C07247=1066.189,109.363,-74.257,172.619,27.910,155.103
C07248=1066.184,109.114,-74.238,172.618,27.907,155.103
C07249=1066.178,108.864,-74.219,172.616,27.904,155.103
C07250=1066.172,108.615,-74.200,172.615,27.901,155.102
C07251=1066.166,108.366,-74.181,172.613,27.898,155.102
C07252=1066.160,108.117,-74.161,172.612,27.896,155.101
C07253=1066.154,107.868,-74.142,172.609,27.893,155.101
C07254=1066.148,107.618,-74.123,172.608,27.890,155.101
C07255=1066.143,107.370,-74.104,172.606,27.887,155.100
C07256=1066.137,107.120,-74.085,172.604,27.885,155.100
C07257=1066.131,106.871,-74.066,172.603,27.882,155.100
C07258=1066.125,106.621,-74.047,172.601,27.879,155.099
C07259=1066.119,106.373,-74.027,172.600,27.877,155.099
C07260=1066.113,106.123,-74.008,172.598,27.874,155.098
C07261=1066.107,105.874,-73.989,172.597,27.871,155.098
C07262=1066.102,105.625,-73.969,172.595,27.868,155.098
C07263=1066.096,105.376,-73.951,172.594,27.865,155.097
C07264=1066.090,105.127,-73.932,172.592,27.863,155.097
C07265=1066.084,104.877,-73.913,172.591,27.860,155.096
C07266=1066.078,104.628,-73.894,172.589,27.857,155.096
C07267=1066.072,104.379,-73.875,172.588,27.854,155.095
C07268=1066.067,104.129,-73.856,172.586,27.852,155.095
C07269=1066.061,103.880,-73.836,172.584,27.849,155.095
C07270=1066.055,103.631,-73.818,172.583,27.847,155.094
C07271=1066.049,103.382,-73.799,172.581,27.844,155.094
C07272=1066.044,103.133,-73.779,172.580,27.841,155.094
C07273=1066.037,102.883,-73.761,172.579,27.838,155.093
C07274=1066.032,102.634,-73.742,172.578,27.836,155.093
C07275=1066.027,102.385,-73.723,172.576,27.833,155.092
C07276=1066.021,102.136,-73.703,172.575,27.830,155.092
C07277=1066.014,101.887,-73.685,172.573,27.827,155.092
C07278=1066.009,101.637,-73.666,172.572,27.825,155.091
C07279=1066.003,101.388,-73.646,172.570,27.822,155.091
C07280=1065.997,101.139,-73.628,172.568,27.819,155.090
C07281=1065.992,100.890,-73.609,172.567,27.816,155.090
C07282=1065.985,100.641,-73.590,172.565,27.813,155.090
C07283=1065.979,100.391,-73.571,172.564,27.811,155.089
C07284=1065.973,100.142,-73.552,172.562,27.808,155.089
C07285=1065.967,99.893,-73.533,172.561,27.806,155.088
C07286=1065.962,99.645,-73.515,172.559,27.803,155.088
C07287=1065.956,99.394,-73.496,172.558,27.800,155.088
C07288=1065.950,99.145,-73.478,172.556,27.797,155.087
C07289=1065.944,98.896,-73.458,172.555,27.794,155.087
C07290=1065.938,98.647,-73.440,172.553,27.792,155.086
C07291=1065.933,98.398,-73.421,172.551,27.789,155.086
C07292=1065.926,98.149,-73.402,172.550,27.787,155.086
C07293=1065.921,97.899,-73.384,172.548,27.784,155.085
C07294=1065.914,97.650,-73.365,172.547,27.781,155.085
C07295=1065.909,97.400,-73.346,172.545,27.778,155.085
C07296=1065.903,97.152,-73.327,172.544,27.775,155.084
C07297=1065.897,96.902,-73.308,172.542,27.773,155.084
C07298=1065.891,96.653,-73.290,172.541,27.770,155.083
C07299=1065.885,96.404,-73.272,172.539,27.767,155.083
C07300=1065.879,96.155,-73.253,172.538,27.765,155.083
C07301=1065.873,95.906,-73.234,172.536,27.762,155.082
C07302=1065.868,95.656,-73.216,172.535,27.759,155.082
C07303=1065.861,95.407,-73.197,172.533,27.756,155.081
C07304=1065.856,95.158,-73.178,172.531,27.754,155.081
C07305=1065.849,94.874,-73.157,172.530,27.751,155.081
C07306=1065.843,94.591,-73.136,172.529,27.748,155.080
C07307=1065.836,94.307,-73.115,172.526,27.745,155.080
C07308=1065.829,94.023,-73.094,172.525,27.741,155.079
C07309=1065.823,93.775,-73.075,172.523,27.738,155.079
C07310=1065.817,93.525,-73.057,172.522,27.736,155.078
C07311=1065.812,93.275,-73.038,172.520,27.733,155.078
C07312=1065.806,93.027,-73.019,172.519,27.730,155.078
C07313=1065.800,92.777,-73.001,172.517,27.728,155.077
C07314=1065.794,92.528,-72.982,172.515,27.725,155.077
C07315=1065.788,92.279,-72.964,172.514,27.722,155.077
C07316=1065.783,92.029,-72.945,172.512,27.719,155.076
C07317=1065.776,91.780,-72.927,172.511,27.717,155.076
C07318=1065.772,91.531,-72.909,172.510,27.714,155.075
C07319=1065.765,91.282,-72.890,172.509,27.711,155.075
C07320=1065.759,91.033,-72.871,172.507,27.708,155.075
C07321=1065.754,90.783,-72.853,172.506,27.706,155.074
C07322=1065.748,90.534,-72.834,172.504,27.703,155.074
C07323=1065.741,90.284,-72.816,172.503,27.700,155.073
C07324=1065.736,90.036,-72.798,172.501,27.697,155.073
C07325=1065.730,89.786,-72.780,172.499,27.695,155.073
C07326=1065.724,89.537,-72.761,172.498,27.692,155.072
C07327=1065.717,89.288,-72.742,172.496,27.689,155.072
C07328=1065.712,89.039,-72.725,172.495,27.687,155.071
C07329=1065.705,88.790,-72.706,172.493,27.684,155.071
C07330=1065.700,88.540,-72.688,172.492,27.681,155.071
C07331=1065.694,88.291,-72.669,172.490,27.679,155.070
C07332=1065.688,88.041,-72.651,172.489,27.676,155.070
C07333=1065.682,87.792,-72.633,172.487,27.673,155.070
C07334=1065.676,87.543,-72.615,172.486,27.670,155.069
C07335=1065.670,87.293,-72.597,172.484,27.668,155.069
C07336=1065.664,87.044,-72.578,172.483,27.665,155.068
C07337=1065.659,86.795,-72.560,172.481,27.663,155.068
C07338=1065.652,86.546,-72.542,172.480,27.660,155.068
C07339=1065.647,86.297,-72.524,172.478,27.657,155.067
C07340=1065.640,86.048,-72.506,172.476,27.654,155.067
C07341=1065.634,85.798,-72.488,172.476,27.652,155.066
C07342=1065.629,85.549,-72.470,172.474,27.649,155.066
C07343=1065.623,85.299,-72.451,172.473,27.646,155.066
C07344=1065.617,85.050,-72.433,172.471,27.643,155.065
C07345=1065.611,84.801,-72.415,172.470,27.641,155.065
C07346=1065.605,84.552,-72.397,172.468,27.638,155.065
C07347=1065.600,84.303,-72.379,172.467,27.635,155.064
C07348=1065.593,84.053,-72.360,172.465,27.633,155.064
C07349=1065.588,83.804,-72.343,172.464,27.630,155.063
C07350=1065.582,83.554,-72.324,172.462,27.627,155.063
C07351=1065.576,83.305,-72.306,172.461,27.624,155.063
C07352=1065.570,83.056,-72.288,172.459,27.621,155.062
C07353=1065.564,82.806,-72.270,172.458,27.619,155.062
C07354=1065.558,82.558,-72.252,172.456,27.616,155.062
C07355=1065.552,82.308,-72.234,172.454,27.614,155.061
C07356=1065.547,82.059,-72.216,172.453,27.611,155.061
C07357=1065.541,81.809,-72.199,172.451,27.608,155.060
C07358=1065.535,81.561,-72.180,172.451,27.605,155.060
C07359=1065.529,81.311,-72.162,172.449,27.603,155.059
C07360=1065.523,81.061,-72.144,172.448,27.600,155.059
C07361=1065.517,80.813,-72.125,172.446,27.597,155.059
C07362=1065.511,80.563,-72.108,172.445,27.594,155.058
C07363=1065.506,80.314,-72.090,172.443,27.591,155.058
C07364=1065.500,80.064,-72.072,172.442,27.589,155.058
C07365=1065.494,79.815,-72.054,172.440,27.586,155.057
C07366=1065.488,79.566,-72.036,172.439,27.583,155.057
C07367=1065.482,79.317,-72.018,172.437,27.581,155.056
C07368=1065.476,79.067,-72.000,172.436,27.578,155.056
C07369=1065.470,78.784,-71.980,172.434,27.575,155.056
C07370=1065.464,78.500,-71.960,172.433,27.572,155.055
C07371=1065.456,78.217,-71.940,172.431,27.568,155.055
C07372=1065.449,77.933,-71.919,172.429,27.565,155.054
C07373=1065.444,77.684,-71.901,172.427,27.563,155.054
C07374=1065.438,77.435,-71.883,172.427,27.560,155.053
C07375=1065.432,77.186,-71.866,172.425,27.557,155.053
C07376=1065.426,76.936,-71.848,172.424,27.555,155.053
C07377=1065.420,76.687,-71.831,172.422,27.552,155.052
C07378=1065.414,76.437,-71.813,172.421,27.549,155.052
C07379=1065.408,76.189,-71.795,172.419,27.547,155.052
C07380=1065.402,75.939,-71.777,172.418,27.544,155.051
C07381=1065.396,75.690,-71.759,172.416,27.541,155.051
C07382=1065.390,75.440,-71.741,172.415,27.539,155.050
C07383=1065.385,75.191,-71.724,172.413,27.536,155.050
C07384=1065.379,74.942,-71.706,172.412,27.533,155.050
C07385=1065.372,74.693,-71.689,172.410,27.530,155.049
C07386=1065.366,74.443,-71.671,172.409,27.527,155.049
C07387=1065.361,74.194,-71.653,172.407,27.525,155.048
C07388=1065.355,73.944,-71.635,172.406,27.522,155.048
C07389=1065.349,73.695,-71.618,172.405,27.520,155.048
C07390=1065.343,73.446,-71.600,172.403,27.517,155.047
C07391=1065.337,73.197,-71.583,172.402,27.514,155.047
C07392=1065.331,72.948,-71.565,172.400,27.511,155.047
C07393=1065.325,72.698,-71.547,172.399,27.509,155.046
C07394=1065.320,72.449,-71.530,172.397,27.506,155.046
C07395=1065.313,72.199,-71.512,172.396,27.503,155.045
C07396=1065.308,71.950,-71.494,172.394,27.500,155.045
C07397=1065.301,71.701,-71.477,172.393,27.498,155.045
C07398=1065.296,71.452,-71.459,172.391,27.495,155.044
C07399=1065.290,71.203,-71.442,172.390,27.492,155.044
C07400=1065.284,70.953,-71.424,172.388,27.489,155.043
C07401=1065.279,70.703,-71.407,172.388,27.487,155.043
C07402=1065.272,70.454,-71.390,172.386,27.484,155.043
C07403=1065.266,70.205,-71.372,172.385,27.481,155.042
C07404=1065.261,69.956,-71.354,172.383,27.479,155.042
C07405=1065.255,69.706,-71.336,172.382,27.476,155.042
C07406=1065.248,69.457,-71.319,172.380,27.473,155.041
C07407=1065.242,69.208,-71.302,172.379,27.471,155.041
C07408=1065.237,68.959,-71.284,172.377,27.468,155.040
C07409=1065.230,68.708,-71.267,172.376,27.465,155.040
C07410=1065.225,68.459,-71.250,172.374,27.463,155.040
C07411=1065.219,68.210,-71.232,172.372,27.460,155.039
C07412=1065.212,67.961,-71.215,172.371,27.457,155.039
C07413=1065.207,67.712,-71.197,172.369,27.454,155.039
C07414=1065.202,67.462,-71.180,172.369,27.452,155.038
C07415=1065.195,67.213,-71.163,172.367,27.449,155.038
C07416=1065.189,66.964,-71.146,172.366,27.447,155.037
C07417=1065.183,66.714,-71.128,172.364,27.444,155.037
C07418=1065.177,66.465,-71.111,172.363,27.441,155.037
C07419=1065.172,66.216,-71.094,172.361,27.438,155.036
C07420=1065.165,65.966,-71.076,172.360,27.435,155.036
C07421=1065.159,65.717,-71.059,172.358,27.433,155.035
C07422=1065.154,65.468,-71.041,172.357,27.430,155.035
C07423=1065.147,65.218,-71.025,172.355,27.428,155.035
C07424=1065.142,64.969,-71.007,172.354,27.425,155.034
C07425=1065.136,64.720,-70.990,172.352,27.422,155.034
C07426=1065.130,64.470,-70.973,172.352,27.419,155.034
C07427=1065.124,64.221,-70.955,172.350,27.417,155.033
C07428=1065.117,63.972,-70.938,172.349,27.414,155.033
C07429=1065.111,63.722,-70.922,172.347,27.411,155.032
C07430=1065.106,63.473,-70.904,172.346,27.409,155.032
C07431=1065.099,63.224,-70.887,172.344,27.406,155.032
C07432=1065.094,62.974,-70.870,172.342,27.404,155.031
C07433=1065.087,62.690,-70.851,172.341,27.401,155.031
C07434=1065.080,62.407,-70.831,172.340,27.397,155.030
C07435=1065.073,62.123,-70.812,172.337,27.394,155.030
C07436=1065.066,61.839,-70.792,172.336,27.391,155.030
C07437=1065.060,61.590,-70.775,172.334,27.389,155.029
C07438=1065.053,61.341,-70.758,172.333,27.386,155.029
C07439=1065.047,61.091,-70.741,172.332,27.384,155.029
C07440=1065.041,60.843,-70.724,172.331,27.381,155.028
C07441=1065.035,60.592,-70.708,172.329,27.378,155.028
C07442=1065.029,60.343,-70.690,172.327,27.376,155.028
C07443=1065.023,60.095,-70.673,172.326,27.373,155.027
C07444=1065.017,59.844,-70.656,172.324,27.370,155.027
C07445=1065.011,59.596,-70.639,172.323,27.368,155.026
C07446=1065.005,59.346,-70.623,172.321,27.365,155.026
C07447=1064.999,59.097,-70.605,172.320,27.362,155.026
C07448=1064.993,58.847,-70.588,172.318,27.360,155.025
C07449=1064.987,58.598,-70.571,172.317,27.357,155.025
C07450=1064.981,58.349,-70.555,172.316,27.355,155.025
C07451=1064.974,58.099,-70.537,172.315,27.352,155.024
C07452=1064.969,57.850,-70.521,172.313,27.349,155.024
C07453=1064.963,57.601,-70.503,172.312,27.346,155.023
C07454=1064.957,57.352,-70.487,172.310,27.344,155.023
C07455=1064.950,57.102,-70.470,172.309,27.341,155.023
C07456=1064.945,56.853,-70.453,172.307,27.338,155.022
C07457=1064.939,56.603,-70.437,172.306,27.336,155.022
C07458=1064.932,56.354,-70.419,172.304,27.333,155.022
C07459=1064.927,56.104,-70.403,172.303,27.331,155.021
C07460=1064.921,55.855,-70.386,172.301,27.328,155.021
C07461=1064.915,55.606,-70.369,172.300,27.325,155.020
C07462=1064.909,55.357,-70.352,172.299,27.322,155.020
C07463=1064.903,55.107,-70.335,172.298,27.320,155.020
C07464=1064.897,54.858,-70.319,172.296,27.317,155.019
C07465=1064.891,54.609,-70.301,172.295,27.314,155.019
C07466=1064.885,54.359,-70.285,172.293,27.312,155.019
C07467=1064.879,54.109,-70.268,172.292,27.309,155.018
C07468=1064.872,53.860,-70.251,172.290,27.307,155.018
C07469=1064.867,53.611,-70.235,172.288,27.304,155.017
C07470=1064.861,53.361,-70.218,172.287,27.301,155.017
C07471=1064.855,53.113,-70.201,172.286,27.298,155.017
C07472=1064.849,52.862,-70.184,172.285,27.296,155.016
C07473=1064.843,52.613,-70.168,172.283,27.293,155.016
C07474=1064.837,52.364,-70.151,172.282,27.290,155.016
C07475=1064.831,52.115,-70.135,172.280,27.288,155.015
C07476=1064.826,51.865,-70.118,172.279,27.285,155.015
C07477=1064.820,51.617,-70.101,172.277,27.282,155.015
C07478=1064.813,51.366,-70.084,172.276,27.280,155.014
C07479=1064.808,51.117,-70.067,172.274,27.277,155.014
C07480=1064.802,50.867,-70.051,172.273,27.274,155.013
C07481=1064.796,50.619,-70.034,172.271,27.271,155.013
C07482=1064.790,50.369,-70.018,172.270,27.269,155.013
C07483=1064.784,50.120,-70.001,172.269,27.266,155.012
C07484=1064.779,49.870,-69.985,172.268,27.264,155.012
C07485=1064.772,49.621,-69.967,172.266,27.261,155.011
C07486=1064.766,49.372,-69.951,172.265,27.258,155.011
C07487=1064.760,49.122,-69.934,172.263,27.256,155.011
C07488=1064.755,48.873,-69.918,172.262,27.253,155.010
C07489=1064.749,48.623,-69.902,172.260,27.250,155.010
C07490=1064.742,48.375,-69.885,172.259,27.247,155.010
C07491=1064.737,48.125,-69.868,172.257,27.244,155.009
C07492=1064.731,47.875,-69.852,172.256,27.241,155.009
C07493=1064.725,47.626,-69.835,172.255,27.239,155.008
C07494=1064.719,47.377,-69.819,172.254,27.237,155.008
C07495=1064.713,47.126,-69.802,172.252,27.234,155.008
C07496=1064.707,46.878,-69.785,172.251,27.231,155.007
C07497=1064.701,46.594,-69.766,172.249,27.228,155.007
C07498=1064.694,46.309,-69.748,172.248,27.225,155.006
C07499=1064.687,46.026,-69.728,172.245,27.222,155.006
C07500=1064.680,45.742,-69.710,172.244,27.219,155.006
C07501=1064.675,45.492,-69.694,172.243,27.216,155.005
C07502=1064.669,45.243,-69.677,172.241,27.213,155.005
C07503=1064.663,44.994,-69.661,172.240,27.210,155.004
C07504=1064.657,44.744,-69.645,172.239,27.208,155.004
C07505=1064.651,44.495,-69.629,172.237,27.205,155.004
C07506=1064.646,44.245,-69.612,172.236,27.203,155.003
C07507=1064.640,43.996,-69.595,172.235,27.200,155.003
C07508=1064.634,43.746,-69.579,172.233,27.197,155.003
C07509=1064.628,43.497,-69.563,172.232,27.194,155.002
C07510=1064.622,43.248,-69.547,172.230,27.192,155.002
C07511=1064.616,42.998,-69.530,172.228,27.189,155.002
C07512=1064.610,42.749,-69.514,172.227,27.186,155.001
C07513=1064.604,42.500,-69.498,172.226,27.183,155.001
C07514=1064.598,42.250,-69.482,172.225,27.181,155.000
C07515=1064.592,42.001,-69.465,172.223,27.179,155.000
C07516=1064.586,41.752,-69.449,172.222,27.176,155.000
C07517=1064.580,41.502,-69.433,172.220,27.173,154.999
C07518=1064.574,41.253,-69.417,172.219,27.171,154.999
C07519=1064.569,41.004,-69.400,172.217,27.168,154.999
C07520=1064.563,40.754,-69.384,172.216,27.165,154.998
C07521=1064.557,40.505,-69.368,172.214,27.163,154.998
C07522=1064.551,40.256,-69.352,172.213,27.160,154.998
C07523=1064.545,40.006,-69.335,172.211,27.157,154.997
C07524=1064.539,39.757,-69.319,172.211,27.154,154.997
C07525=1064.533,39.508,-69.303,172.209,27.152,154.996
C07526=1064.527,39.258,-69.287,172.208,27.149,154.996
C07527=1064.521,39.008,-69.271,172.206,27.146,154.996
C07528=1064.515,38.759,-69.255,172.205,27.144,154.995
C07529=1064.509,38.510,-69.238,172.203,27.141,154.995
C07530=1064.503,38.260,-69.222,172.202,27.139,154.995
C07531=1064.497,38.011,-69.206,172.200,27.136,154.994
C07532=1064.491,37.761,-69.190,172.199,27.133,154.994
C07533=1064.485,37.512,-69.174,172.197,27.131,154.993
C07534=1064.479,37.262,-69.159,172.197,27.128,154.993
C07535=1064.473,37.013,-69.142,172.195,27.126,154.993
C07536=1064.467,36.764,-69.126,172.194,27.123,154.992
C07537=1064.461,36.514,-69.110,172.192,27.120,154.992
C07538=1064.455,36.265,-69.094,172.191,27.118,154.992
C07539=1064.449,36.015,-69.079,172.189,27.115,154.991
C07540=1064.443,35.766,-69.062,172.188,27.112,154.991
C07541=1064.437,35.517,-69.046,172.186,27.110,154.991
C07542=1064.430,35.268,-69.030,172.185,27.107,154.990
C07543=1064.425,35.018,-69.015,172.183,27.105,154.990
C07544=1064.419,34.768,-68.999,172.182,27.102,154.990
C07545=1064.413,34.519,-68.982,172.181,27.099,154.989
C07546=1064.406,34.270,-68.967,172.180,27.097,154.989
C07547=1064.400,34.020,-68.951,172.178,27.094,154.989
C07548=1064.395,33.771,-68.935,172.177,27.091,154.988
C07549=1064.389,33.521,-68.919,172.175,27.089,154.988
C07550=1064.382,33.272,-68.904,172.174,27.086,154.987
C07551=1064.376,33.022,-68.887,172.172,27.083,154.987
C07552=1064.370,32.773,-68.871,172.171,27.081,154.987
C07553=1064.365,32.523,-68.856,172.169,27.078,154.986
C07554=1064.358,32.274,-68.840,172.168,27.075,154.986
C07555=1064.352,32.025,-68.824,172.166,27.073,154.986
C07556=1064.346,31.775,-68.808,172.166,27.071,154.985
C07557=1064.340,31.525,-68.792,172.164,27.068,154.985
C07558=1064.334,31.277,-68.777,172.163,27.065,154.985
C07559=1064.329,31.027,-68.761,172.161,27.063,154.984
C07560=1064.323,30.778,-68.745,172.160,27.060,154.984
C07561=1064.315,30.494,-68.727,172.158,27.057,154.983
C07562=1064.309,30.209,-68.709,172.157,27.054,154.983
C07563=1064.302,29.925,-68.691,172.154,27.051,154.983
C07564=1064.295,29.642,-68.673,172.153,27.048,154.982
C07565=1064.290,29.392,-68.658,172.151,27.045,154.982
C07566=1064.283,29.143,-68.642,172.150,27.042,154.982
C07567=1064.277,28.894,-68.626,172.149,27.040,154.981
C07568=1064.271,28.644,-68.610,172.148,27.038,154.981
C07569=1064.265,28.395,-68.595,172.146,27.035,154.981
C07570=1064.259,28.145,-68.579,172.145,27.032,154.980
C07571=1064.254,27.896,-68.563,172.143,27.030,154.980
C07572=1064.247,27.646,-68.548,172.142,27.027,154.979
C07573=1064.241,27.397,-68.532,172.140,27.025,154.979
C07574=1064.235,27.147,-68.517,172.139,27.022,154.979
C07575=1064.229,26.898,-68.501,172.137,27.019,154.978
C07576=1064.223,26.648,-68.486,172.136,27.017,154.978
C07577=1064.217,26.399,-68.469,172.134,27.014,154.978
C07578=1064.211,26.149,-68.454,172.134,27.012,154.977
C07579=1064.205,25.901,-68.439,172.132,27.009,154.977
C07580=1064.199,25.651,-68.423,172.131,27.007,154.977
C07581=1064.193,25.401,-68.408,172.129,27.004,154.976
C07582=1064.187,25.152,-68.392,172.128,27.001,154.976
C07583=1064.181,24.902,-68.377,172.126,26.999,154.976
C07584=1064.175,24.653,-68.361,172.125,26.996,154.975
C07585=1064.168,24.403,-68.346,172.123,26.993,154.975
C07586=1064.163,24.154,-68.331,172.122,26.991,154.975
C07587=1064.157,23.905,-68.315,172.120,26.988,154.974
C07588=1064.151,23.655,-68.299,172.119,26.986,154.974
C07589=1064.144,23.406,-68.284,172.118,26.983,154.974
C07590=1064.139,23.156,-68.268,172.117,26.981,154.973
C07591=1064.133,22.907,-68.254,172.115,26.978,154.973
C07592=1064.127,22.657,-68.237,172.114,26.976,154.973
C07593=1064.121,22.408,-68.222,172.112,26.973,154.972
C07594=1064.115,22.158,-68.207,172.111,26.970,154.972
C07595=1064.108,21.909,-68.191,172.109,26.968,154.972
C07596=1064.103,21.659,-68.176,172.108,26.965,154.971
C07597=1064.097,21.410,-68.161,172.106,26.963,154.971
C07598=1064.090,21.161,-68.145,172.105,26.960,154.971
C07599=1064.084,20.911,-68.130,172.103,26.957,154.970
C07600=1064.078,20.661,-68.115,172.102,26.955,154.970
C07601=1064.073,20.413,-68.099,172.101,26.952,154.969
C07602=1064.066,20.163,-68.084,172.099,26.950,154.969
C07603=1064.061,19.913,-68.069,172.098,26.947,154.969
C07604=1064.054,19.663,-68.054,172.096,26.945,154.969
C07605=1064.048,19.415,-68.038,172.095,26.942,154.968
C07606=1064.043,19.165,-68.023,172.093,26.940,154.968
C07607=1064.036,18.915,-68.008,172.092,26.937,154.967
C07608=1064.030,18.666,-67.993,172.090,26.935,154.967
C07609=1064.024,18.416,-67.977,172.089,26.932,154.967
C07610=1064.018,18.167,-67.962,172.087,26.930,154.967
C07611=1064.012,17.917,-67.946,172.086,26.927,154.966
C07612=1064.006,17.668,-67.932,172.085,26.925,154.966
C07613=1064.000,17.419,-67.917,172.084,26.922,154.965
C07614=1063.995,17.169,-67.901,172.082,26.920,154.965
C07615=1063.988,16.920,-67.886,172.081,26.917,154.965
C07616=1063.982,16.670,-67.871,172.079,26.914,154.964
C07617=1063.976,16.421,-67.856,172.078,26.912,154.964
C07618=1063.970,16.171,-67.841,172.076,26.909,154.964
C07619=1063.964,15.921,-67.826,172.075,26.906,154.963
C07620=1063.958,15.672,-67.810,172.073,26.904,154.963
C07621=1063.952,15.423,-67.795,172.072,26.901,154.963
C07622=1063.946,15.174,-67.780,172.070,26.899,154.963
C07623=1063.939,14.924,-67.765,172.069,26.896,154.962
C07624=1063.934,14.675,-67.750,172.067,26.894,154.962
C07625=1063.927,14.392,-67.733,172.066,26.891,154.961
C07626=1063.920,14.110,-67.716,172.064,26.888,154.961
C07627=1063.913,13.826,-67.698,172.063,26.885,154.961
C07628=1063.907,13.544,-67.682,172.061,26.882,154.960
C07629=1063.900,13.295,-67.667,172.060,26.880,154.960
C07630=1063.894,13.045,-67.652,172.058,26.877,154.960
C07631=1063.887,12.795,-67.637,172.057,26.875,154.959
C07632=1063.882,12.546,-67.622,172.055,26.873,154.959
C07633=1063.875,12.297,-67.607,172.054,26.870,154.959
C07634=1063.869,12.047,-67.592,172.052,26.868,154.958
C07635=1063.863,11.798,-67.578,172.051,26.865,154.958
C07636=1063.857,11.548,-67.562,172.049,26.862,154.958
C07637=1063.851,11.298,-67.547,172.048,26.860,154.957
C07638=1063.845,11.049,-67.532,172.047,26.858,154.957
C07639=1063.839,10.800,-67.518,172.046,26.855,154.957
C07640=1063.833,10.550,-67.503,172.044,26.853,154.957
C07641=1063.826,10.301,-67.488,172.043,26.850,154.956
C07642=1063.820,10.052,-67.473,172.041,26.848,154.956
C07643=1063.814,9.802,-67.458,172.040,26.846,154.956
C07644=1063.808,9.552,-67.444,172.038,26.843,154.955
C07645=1063.802,9.303,-67.430,172.037,26.840,154.955
C07646=1063.796,9.053,-67.415,172.035,26.838,154.955
C07647=1063.789,8.803,-67.400,172.034,26.835,154.954
C07648=1063.784,8.554,-67.385,172.032,26.833,154.954
C07649=1063.778,8.304,-67.370,172.031,26.830,154.954
C07650=1063.772,8.055,-67.355,172.029,26.828,154.953
C07651=1063.766,7.806,-67.340,172.028,26.826,154.953
C07652=1063.759,7.556,-67.325,172.026,26.823,154.953
C07653=1063.754,7.307,-67.311,172.025,26.821,154.952
C07654=1063.748,7.057,-67.296,172.024,26.818,154.952
C07655=1063.741,6.807,-67.281,172.022,26.816,154.952
C07656=1063.735,6.558,-67.267,172.021,26.813,154.951
C07657=1063.729,6.309,-67.252,172.019,26.810,154.951
C07658=1063.723,6.060,-67.237,172.018,26.808,154.951
C07659=1063.717,5.810,-67.222,172.016,26.806,154.951
C07660=1063.711,5.560,-67.208,172.015,26.803,154.950
C07661=1063.705,5.311,-67.193,172.013,26.801,154.950
C07662=1063.699,5.061,-67.179,172.012,26.798,154.950
C07663=1063.693,4.812,-67.164,172.010,26.795,154.949
C07664=1063.686,4.563,-67.149,172.009,26.793,154.949
C07665=1063.681,4.313,-67.135,172.007,26.790,154.949
C07666=1063.675,4.063,-67.120,172.006,26.788,154.948
C07667=1063.668,3.814,-67.105,172.005,26.786,154.948
C07668=1063.662,3.565,-67.091,172.004,26.783,154.948
C07669=1063.656,3.314,-67.076,172.002,26.781,154.947
C07670=1063.650,3.066,-67.062,172.001,26.779,154.947
C07671=1063.644,2.816,-67.047,171.999,26.776,154.947
C07672=1063.639,2.566,-67.033,171.998,26.773,154.946
C07673=1063.632,2.317,-67.018,171.996,26.771,154.946
C07674=1063.626,2.068,-67.004,171.995,26.768,154.946
C07675=1063.620,1.818,-66.989,171.993,26.766,154.945
C07676=1063.615,1.568,-66.975,171.992,26.763,154.945
C07677=1063.608,1.319,-66.960,171.990,26.761,154.945
C07678=1063.602,1.070,-66.945,171.989,26.759,154.945
C07679=1063.596,0.820,-66.931,171.987,26.756,154.944
C07680=1063.591,0.571,-66.916,171.986,26.753,154.944
C07681=1063.584,0.321,-66.901,171.984,26.751,154.944
C07682=1063.579,0.071,-66.888,171.983,26.748,154.943
C07683=1063.572,-0.178,-66.873,171.982,26.746,154.943
C07684=1063.567,-0.428,-66.859,171.981,26.744,154.943
C07685=1063.560,-0.678,-66.844,171.979,26.741,154.942
C07686=1063.555,-0.926,-66.829,171.978,26.739,154.942
C07687=1063.549,-1.177,-66.815,171.976,26.736,154.942
C07688=1063.543,-1.426,-66.800,171.975,26.734,154.941
C07689=1063.537,-1.707,-66.784,171.973,26.731,154.941
C07690=1063.529,-1.988,-66.768,171.971,26.728,154.941
C07691=1063.523,-2.267,-66.752,171.969,26.725,154.940
C07692=1063.516,-2.548,-66.736,171.968,26.722,154.940
C07693=1063.510,-2.797,-66.721,171.966,26.720,154.940
C07694=1063.504,-3.048,-66.707,171.965,26.718,154.939
C07695=1063.498,-3.297,-66.692,171.963,26.715,154.939
C07696=1063.492,-3.547,-66.678,171.962,26.713,154.939
C07697=1063.486,-3.796,-66.664,171.960,26.710,154.938
C07698=1063.480,-4.046,-66.650,171.959,26.708,154.938
C07699=1063.474,-4.295,-66.635,171.957,26.706,154.938
C07700=1063.468,-4.545,-66.621,171.957,26.703,154.937
C07701=1063.462,-4.794,-66.607,171.955,26.701,154.937
C07702=1063.455,-5.044,-66.593,171.954,26.699,154.937
C07703=1063.449,-5.293,-66.578,171.952,26.696,154.937
C07704=1063.443,-5.543,-66.564,171.950,26.694,154.936
C07705=1063.437,-5.793,-66.551,171.949,26.692,154.936
C07706=1063.431,-6.042,-66.536,171.947,26.689,154.936
C07707=1063.425,-6.292,-66.522,171.946,26.686,154.935
C07708=1063.419,-6.540,-66.508,171.944,26.684,154.935
C07709=1063.413,-6.791,-66.494,171.943,26.682,154.935
C07710=1063.407,-7.040,-66.479,171.941,26.680,154.935
C07711=1063.400,-7.290,-66.466,171.940,26.677,154.934
C07712=1063.394,-7.539,-66.452,171.938,26.674,154.934
C07713=1063.388,-7.789,-66.437,171.937,26.672,154.934
C07714=1063.382,-8.038,-66.424,171.935,26.670,154.933
C07715=1063.376,-8.287,-66.409,171.934,26.668,154.933
C07716=1063.370,-8.537,-66.395,171.932,26.665,154.933
C07717=1063.364,-8.787,-66.381,171.931,26.663,154.933
C07718=1063.357,-9.036,-66.367,171.929,26.660,154.932
C07719=1063.352,-9.286,-66.353,171.928,26.658,154.932
C07720=1063.346,-9.535,-66.339,171.926,26.655,154.932
C07721=1063.339,-9.785,-66.324,171.925,26.653,154.931
C07722=1063.334,-10.034,-66.311,171.924,26.651,154.931
C07723=1063.327,-10.284,-66.297,171.922,26.649,154.931
C07724=1063.322,-10.534,-66.283,171.921,26.647,154.931
C07725=1063.316,-10.783,-66.268,171.919,26.644,154.930
C07726=1063.309,-11.033,-66.255,171.918,26.641,154.930
C07727=1063.304,-11.282,-66.241,171.916,26.639,154.930
C07728=1063.297,-11.531,-66.227,171.915,26.637,154.929
C07729=1063.291,-11.781,-66.213,171.913,26.634,154.929
C07730=1063.285,-12.031,-66.199,171.912,26.632,154.929
C07731=1063.279,-12.280,-66.186,171.910,26.630,154.929
C07732=1063.273,-12.530,-66.171,171.909,26.628,154.928
C07733=1063.267,-12.779,-66.157,171.907,26.625,154.928
C07734=1063.261,-13.029,-66.144,171.906,26.622,154.928
C07735=1063.255,-13.279,-66.129,171.904,26.620,154.927
C07736=1063.249,-13.528,-66.116,171.903,26.618,154.927
C07737=1063.243,-13.777,-66.101,171.901,26.615,154.927
C07738=1063.237,-14.027,-66.087,171.900,26.613,154.927
C07739=1063.231,-14.277,-66.074,171.898,26.611,154.926
C07740=1063.225,-14.526,-66.060,171.896,26.609,154.926
C07741=1063.219,-14.776,-66.046,171.895,26.606,154.926
C07742=1063.213,-15.025,-66.032,171.894,26.603,154.925
C07743=1063.207,-15.274,-66.019,171.892,26.601,154.925
C07744=1063.200,-15.525,-66.004,171.890,26.599,154.925
C07745=1063.194,-15.774,-65.991,171.889,26.596,154.925
C07746=1063.189,-16.024,-65.977,171.887,26.594,154.924
C07747=1063.182,-16.273,-65.964,171.886,26.592,154.924
C07748=1063.176,-16.523,-65.950,171.884,26.590,154.924
C07749=1063.170,-16.772,-65.936,171.883,26.587,154.924
C07750=1063.164,-17.022,-65.923,171.882,26.585,154.923
C07751=1063.158,-17.271,-65.908,171.881,26.583,154.923
C07752=1063.151,-17.521,-65.895,171.879,26.581,154.923
C07753=1063.145,-17.799,-65.880,171.877,26.578,154.923
C07754=1063.138,-18.079,-65.865,171.875,26.576,154.922
C07755=1063.131,-18.358,-65.850,171.874,26.573,154.922
C07756=1063.124,-18.637,-65.835,171.872,26.571,154.922
C07757=1063.118,-18.887,-65.821,171.871,26.568,154.921
C07758=1063.112,-19.136,-65.807,171.869,26.566,154.921
C07759=1063.106,-19.386,-65.793,171.868,26.564,154.921
C07760=1063.100,-19.635,-65.780,171.866,26.561,154.921
C07761=1063.093,-19.885,-65.767,171.864,26.559,154.920
C07762=1063.088,-20.135,-65.753,171.863,26.557,154.920
C07763=1063.082,-20.384,-65.739,171.861,26.554,154.920
C07764=1063.075,-20.633,-65.726,171.860,26.553,154.920
C07765=1063.069,-20.884,-65.712,171.858,26.550,154.919
C07766=1063.063,-21.133,-65.699,171.857,26.548,154.919
C07767=1063.058,-21.382,-65.685,171.855,26.546,154.919
C07768=1063.051,-21.632,-65.672,171.854,26.543,154.919
C07769=1063.045,-21.882,-65.658,171.852,26.541,154.918
C07770=1063.039,-22.131,-65.644,171.851,26.539,154.918
C07771=1063.033,-22.380,-65.631,171.849,26.537,154.918
C07772=1063.027,-22.630,-65.618,171.848,26.534,154.917
C07773=1063.021,-22.879,-65.604,171.846,26.532,154.917
C07774=1063.014,-23.129,-65.590,171.844,26.530,154.917
C07775=1063.008,-23.379,-65.577,171.843,26.527,154.917
C07776=1063.003,-23.629,-65.564,171.841,26.525,154.916
C07777=1062.997,-23.878,-65.550,171.840,26.523,154.916
C07778=1062.991,-24.127,-65.537,171.838,26.520,154.916
C07779=1062.985,-24.377,-65.523,171.837,26.518,154.916
C07780=1062.978,-24.627,-65.510,171.835,26.516,154.915
C07781=1062.972,-24.876,-65.496,171.834,26.514,154.915
C07782=1062.966,-25.125,-65.483,171.832,26.512,154.915
C07783=1062.961,-25.376,-65.470,171.831,26.509,154.915
C07784=1062.954,-25.625,-65.457,171.829,26.507,154.914
C07785=1062.948,-25.874,-65.443,171.827,26.505,154.914
C07786=1062.942,-26.124,-65.429,171.826,26.502,154.914
C07787=1062.936,-26.374,-65.416,171.824,26.500,154.914
C07788=1062.930,-26.623,-65.403,171.823,26.498,154.913
C07789=1062.925,-26.873,-65.389,171.821,26.496,154.913
C07790=1062.918,-27.122,-65.376,171.820,26.494,154.913
C07791=1062.912,-27.372,-65.363,171.818,26.491,154.913
C07792=1062.905,-27.622,-65.349,171.817,26.489,154.912
C07793=1062.899,-27.871,-65.337,171.815,26.487,154.912
C07794=1062.893,-28.121,-65.323,171.814,26.485,154.912
C07795=1062.887,-28.370,-65.310,171.812,26.483,154.912
C07796=1062.881,-28.619,-65.297,171.810,26.480,154.911
C07797=1062.875,-28.869,-65.284,171.809,26.478,154.911
C07798=1062.869,-29.118,-65.271,171.807,26.476,154.911
C07799=1062.863,-29.369,-65.257,171.806,26.474,154.911
C07800=1062.857,-29.619,-65.244,171.804,26.472,154.910
C07801=1062.850,-29.868,-65.231,171.803,26.470,154.910
C07802=1062.844,-30.117,-65.218,171.801,26.468,154.910
C07803=1062.838,-30.367,-65.205,171.800,26.465,154.910
C07804=1062.832,-30.616,-65.192,171.798,26.463,154.910
C07805=1062.826,-30.865,-65.179,171.796,26.461,154.909
C07806=1062.819,-31.116,-65.166,171.795,26.459,154.909
C07807=1062.813,-31.365,-65.152,171.793,26.457,154.909
C07808=1062.807,-31.615,-65.139,171.792,26.454,154.909
C07809=1062.801,-31.864,-65.127,171.790,26.452,154.908
C07810=1062.795,-32.114,-65.113,171.789,26.450,154.908
C07811=1062.789,-32.364,-65.101,171.787,26.448,154.908
C07812=1062.783,-32.613,-65.088,171.786,26.446,154.908
C07813=1062.776,-32.862,-65.074,171.784,26.444,154.907
C07814=1062.771,-33.112,-65.061,171.782,26.442,154.907
C07815=1062.765,-33.362,-65.048,171.781,26.439,154.907
C07816=1062.759,-33.611,-65.035,171.779,26.437,154.907
C07817=1062.752,-33.890,-65.021,171.778,26.435,154.906
C07818=1062.745,-34.168,-65.006,171.776,26.432,154.906
C07819=1062.738,-34.446,-64.991,171.775,26.430,154.906
C07820=1062.731,-34.724,-64.977,171.773,26.428,154.906
C07821=1062.725,-34.974,-64.965,171.772,26.426,154.905
C07822=1062.720,-35.224,-64.951,171.770,26.424,154.905
C07823=1062.714,-35.473,-64.938,171.769,26.421,154.905
C07824=1062.708,-35.723,-64.925,171.767,26.420,154.905
C07825=1062.702,-35.973,-64.912,171.765,26.417,154.905
C07826=1062.695,-36.222,-64.899,171.763,26.415,154.904
C07827=1062.690,-36.472,-64.887,171.761,26.413,154.904
C07828=1062.683,-36.721,-64.873,171.760,26.411,154.904
C07829=1062.677,-36.971,-64.861,171.758,26.408,154.904
C07830=1062.671,-37.220,-64.848,171.757,26.407,154.904
C07831=1062.665,-37.470,-64.835,171.755,26.404,154.903
C07832=1062.659,-37.719,-64.822,171.754,26.402,154.903
C07833=1062.653,-37.969,-64.809,171.752,26.400,154.903
C07834=1062.647,-38.219,-64.797,171.750,26.398,154.903
C07835=1062.641,-38.468,-64.783,171.749,26.396,154.902
C07836=1062.635,-38.718,-64.771,171.747,26.394,154.902
C07837=1062.628,-38.967,-64.758,171.746,26.392,154.902
C07838=1062.622,-39.217,-64.746,171.744,26.390,154.902
C07839=1062.616,-39.467,-64.733,171.743,26.388,154.901
C07840=1062.610,-39.716,-64.720,171.741,26.386,154.901
C07841=1062.604,-39.966,-64.707,171.739,26.384,154.901
C07842=1062.598,-40.216,-64.695,171.738,26.382,154.901
C07843=1062.591,-40.465,-64.682,171.736,26.379,154.901
C07844=1062.585,-40.715,-64.669,171.735,26.378,154.901
C07845=1062.579,-40.964,-64.656,171.733,26.375,154.900
C07846=1062.573,-41.214,-64.644,171.731,26.374,154.900
C07847=1062.567,-41.463,-64.632,171.730,26.371,154.900
C07848=1062.561,-41.713,-64.619,171.728,26.370,154.900
C07849=1062.555,-41.963,-64.606,171.727,26.367,154.899
C07850=1062.549,-42.213,-64.593,171.725,26.366,154.899
C07851=1062.542,-42.462,-64.581,171.724,26.363,154.899
C07852=1062.536,-42.711,-64.568,171.722,26.361,154.899
C07853=1062.530,-42.961,-64.555,171.720,26.359,154.899
C07854=1062.524,-43.211,-64.543,171.719,26.357,154.898
C07855=1062.518,-43.461,-64.530,171.717,26.355,154.898
C07856=1062.511,-43.710,-64.518,171.716,26.353,154.898
C07857=1062.505,-43.960,-64.505,171.714,26.351,154.898
C07858=1062.499,-44.210,-64.493,171.713,26.349,154.898
C07859=1062.494,-44.459,-64.480,171.711,26.347,154.897
C07860=1062.487,-44.708,-64.468,171.709,26.345,154.897
C07861=1062.481,-44.958,-64.455,171.708,26.343,154.897
C07862=1062.475,-45.208,-64.443,171.706,26.341,154.897
C07863=1062.469,-45.457,-64.430,171.705,26.339,154.897
C07864=1062.463,-45.707,-64.418,171.703,26.337,154.896
C07865=1062.456,-45.956,-64.405,171.701,26.335,154.896
C07866=1062.451,-46.206,-64.392,171.700,26.333,154.896
C07867=1062.445,-46.456,-64.380,171.698,26.331,154.896
C07868=1062.438,-46.706,-64.368,171.697,26.329,154.896
C07869=1062.433,-46.955,-64.356,171.695,26.327,154.895
C07870=1062.427,-47.205,-64.343,171.694,26.325,154.895
C07871=1062.420,-47.454,-64.330,171.692,26.323,154.895
C07872=1062.414,-47.704,-64.318,171.690,26.321,154.895
C07873=1062.408,-47.953,-64.305,171.689,26.319,154.895
C07874=1062.402,-48.203,-64.293,171.687,26.317,154.895
C07875=1062.395,-48.453,-64.281,171.686,26.315,154.894
C07876=1062.390,-48.702,-64.269,171.684,26.313,154.894
C07877=1062.384,-48.952,-64.256,171.682,26.312,154.894
C07878=1062.378,-49.202,-64.244,171.681,26.309,154.894
C07879=1062.372,-49.451,-64.231,171.679,26.307,154.894
C07880=1062.366,-49.701,-64.219,171.678,26.305,154.893
C07881=1062.359,-49.980,-64.205,171.675,26.303,154.893
C07882=1062.352,-50.259,-64.192,171.674,26.301,154.893
C07883=1062.345,-50.536,-64.178,171.672,26.299,154.893
C07884=1062.338,-50.815,-64.164,171.671,26.297,154.893
C07885=1062.333,-51.065,-64.152,171.669,26.295,154.892
C07886=1062.326,-51.314,-64.140,171.666,26.293,154.892
C07887=1062.319,-51.564,-64.128,171.665,26.291,154.892
C07888=1062.313,-51.814,-64.115,171.663,26.289,154.892
C07889=1062.307,-52.063,-64.103,171.662,26.287,154.892
C07890=1062.301,-52.313,-64.091,171.660,26.285,154.892
C07891=1062.294,-52.563,-64.079,171.658,26.284,154.891
C07892=1062.289,-52.813,-64.067,171.657,26.282,154.891
C07893=1062.282,-53.062,-64.055,171.655,26.280,154.891
C07894=1062.276,-53.312,-64.043,171.653,26.278,154.891
C07895=1062.270,-53.562,-64.031,171.652,26.276,154.891
C07896=1062.263,-53.811,-64.019,171.650,26.274,154.891
C07897=1062.257,-54.061,-64.006,171.649,26.273,154.890
C07898=1062.251,-54.311,-63.994,171.647,26.271,154.890
C07899=1062.245,-54.559,-63.983,171.645,26.269,154.890
C07900=1062.239,-54.809,-63.970,171.644,26.267,154.890
C07901=1062.232,-55.059,-63.958,171.642,26.265,154.890
C07902=1062.225,-55.308,-63.946,171.641,26.263,154.890
C07903=1062.220,-55.559,-63.934,171.639,26.262,154.889
C07904=1062.214,-55.808,-63.923,171.637,26.260,154.889
C07905=1062.208,-56.058,-63.910,171.636,26.258,154.889
C07906=1062.201,-56.307,-63.898,171.634,26.256,154.889
C07907=1062.195,-56.557,-63.886,171.632,26.255,154.889
C07908=1062.189,-56.807,-63.874,171.631,26.253,154.889
C07909=1062.183,-57.056,-63.862,171.629,26.250,154.889
C07910=1062.176,-57.306,-63.851,171.628,26.249,154.888
C07911=1062.170,-57.556,-63.838,171.626,26.247,154.888
C07912=1062.164,-57.805,-63.826,171.624,26.245,154.888
C07913=1062.158,-58.054,-63.815,171.622,26.243,154.888
C07914=1062.152,-58.304,-63.802,171.620,26.241,154.888
C07915=1062.146,-58.554,-63.791,171.619,26.240,154.888
C07916=1062.139,-58.804,-63.779,171.617,26.238,154.888
C07917=1062.134,-59.053,-63.767,171.615,26.236,154.887
C07918=1062.127,-59.303,-63.755,171.614,26.234,154.887
C07919=1062.121,-59.553,-63.744,171.612,26.233,154.887
C07920=1062.115,-59.803,-63.731,171.610,26.231,154.887
C07921=1062.109,-60.051,-63.719,171.609,26.229,154.887
C07922=1062.102,-60.301,-63.707,171.607,26.227,154.887
C07923=1062.096,-60.552,-63.696,171.606,26.225,154.886
C07924=1062.090,-60.800,-63.684,171.604,26.223,154.886
C07925=1062.084,-61.050,-63.672,171.602,26.222,154.886
C07926=1062.078,-61.301,-63.660,171.601,26.220,154.886
C07927=1062.071,-61.550,-63.648,171.599,26.218,154.886
C07928=1062.065,-61.799,-63.637,171.597,26.216,154.886
C07929=1062.060,-62.049,-63.625,171.596,26.215,154.886
C07930=1062.053,-62.299,-63.613,171.594,26.213,154.885
C07931=1062.047,-62.548,-63.601,171.593,26.211,154.885
C07932=1062.041,-62.798,-63.589,171.591,26.209,154.885
C07933=1062.035,-63.048,-63.577,171.589,26.208,154.885
C07934=1062.029,-63.297,-63.566,171.588,26.206,154.885
C07935=1062.022,-63.547,-63.555,171.586,26.204,154.885
C07936=1062.017,-63.796,-63.542,171.584,26.202,154.885
C07937=1062.010,-64.046,-63.530,171.582,26.200,154.885
C07938=1062.004,-64.296,-63.519,171.580,26.199,154.884
C07939=1061.999,-64.545,-63.507,171.579,26.197,154.884
C07940=1061.993,-64.795,-63.496,171.577,26.195,154.884
C07941=1061.986,-65.045,-63.484,171.575,26.193,154.884
C07942=1061.980,-65.294,-63.472,171.574,26.192,154.884
C07943=1061.974,-65.544,-63.460,171.572,26.190,154.884
C07944=1061.968,-65.793,-63.449,171.570,26.188,154.884
C07945=1061.959,-66.139,-63.433,171.568,26.186,154.883
C07946=1061.951,-66.484,-63.416,171.566,26.184,154.883
C07947=1061.942,-66.830,-63.401,171.564,26.181,154.883
C07948=1061.935,-67.175,-63.385,171.561,26.179,154.883
C07949=1061.928,-67.425,-63.373,171.560,26.177,154.883
C07950=1061.923,-67.674,-63.362,171.558,26.176,154.883
C07951=1061.916,-67.924,-63.350,171.557,26.174,154.882
C07952=1061.910,-68.174,-63.339,171.555,26.172,154.882
C07953=1061.904,-68.423,-63.326,171.553,26.170,154.882
C07954=1061.898,-68.673,-63.315,171.552,26.169,154.882
C07955=1061.892,-68.922,-63.304,171.550,26.167,154.882
C07956=1061.886,-69.172,-63.292,171.547,26.165,154.882
C07957=1061.880,-69.422,-63.280,171.546,26.164,154.882
C07958=1061.874,-69.672,-63.269,171.544,26.162,154.882
C07959=1061.868,-69.921,-63.257,171.542,26.160,154.881
C07960=1061.862,-70.171,-63.246,171.541,26.158,154.881
C07961=1061.857,-70.421,-63.235,171.539,26.157,154.881
C07962=1061.850,-70.670,-63.223,171.538,26.155,154.881
C07963=1061.844,-70.920,-63.212,171.536,26.153,154.881
C07964=1061.838,-71.169,-63.200,171.534,26.151,154.881
C07965=1061.832,-71.419,-63.189,171.533,26.150,154.881
C07966=1061.826,-71.669,-63.177,171.531,26.148,154.881
C07967=1061.820,-71.918,-63.165,171.529,26.147,154.880
C07968=1061.814,-72.168,-63.154,171.528,26.145,154.880
C07969=1061.808,-72.418,-63.143,171.526,26.143,154.880
C07970=1061.801,-72.667,-63.131,171.524,26.141,154.880
C07971=1061.796,-72.917,-63.120,171.523,26.140,154.880
C07972=1061.790,-73.167,-63.109,171.521,26.138,154.880
C07973=1061.784,-73.416,-63.097,171.519,26.137,154.880
C07974=1061.778,-73.666,-63.086,171.518,26.135,154.880
C07975=1061.772,-73.916,-63.075,171.516,26.133,154.879
C07976=1061.765,-74.165,-63.063,171.514,26.132,154.879
C07977=1061.760,-74.415,-63.052,171.512,26.130,154.879
C07978=1061.753,-74.665,-63.041,171.510,26.128,154.879
C07979=1061.747,-74.914,-63.029,171.509,26.127,154.879
C07980=1061.741,-75.164,-63.018,171.507,26.125,154.879
C07981=1061.735,-75.414,-63.007,171.505,26.124,154.879
C07982=1061.729,-75.664,-62.996,171.504,26.122,154.879
C07983=1061.723,-75.913,-62.984,171.502,26.121,154.879
C07984=1061.716,-76.163,-62.973,171.500,26.119,154.879
C07985=1061.711,-76.412,-62.962,171.499,26.118,154.879
C07986=1061.705,-76.662,-62.951,171.497,26.116,154.878
C07987=1061.699,-76.912,-62.940,171.495,26.114,154.878
C07988=1061.692,-77.161,-62.928,171.494,26.113,154.878
C07989=1061.686,-77.411,-62.917,171.492,26.111,154.878
C07990=1061.680,-77.661,-62.906,171.490,26.110,154.878
C07991=1061.674,-77.911,-62.895,171.489,26.108,154.878
C07992=1061.668,-78.160,-62.884,171.487,26.107,154.878
C07993=1061.662,-78.410,-62.872,171.485,26.105,154.878
C07994=1061.656,-78.659,-62.861,171.484,26.104,154.878
C07995=1061.649,-78.909,-62.851,171.481,26.102,154.878
C07996=1061.643,-79.159,-62.840,171.479,26.100,154.878
C07997=1061.637,-79.408,-62.829,171.478,26.099,154.877
C07998=1061.631,-79.658,-62.818,171.476,26.097,154.877
C07999=1061.625,-79.908,-62.807,171.474,26.096,154.877
C08000=1061.619,-80.158,-62.796,171.473,26.095,154.877
C08001=1061.613,-80.375,-62.786,171.471,26.093,154.877
C08002=1061.608,-80.592,-62.777,171.470,26.092,154.877
C08003=1061.603,-80.809,-62.768,171.468,26.091,154.877
C08004=1061.598,-81.025,-62.757,171.467,26.090,154.877
C08005=1061.592,-81.243,-62.748,171.465,26.088,154.877
C08006=1061.586,-81.460,-62.739,171.463,26.087,154.877
C08007=1061.581,-81.676,-62.729,171.462,26.086,154.877
C08008=1061.575,-81.893,-62.720,171.461,26.085,154.877
C08009=1061.568,-82.176,-62.707,171.459,26.083,154.877
C08010=1061.562,-82.458,-62.695,171.456,26.081,154.877
C08011=1061.554,-82.740,-62.682,171.455,26.080,154.876
C08012=1061.548,-83.022,-62.671,171.453,26.078,154.876
C08013=1061.541,-83.273,-62.660,171.450,26.076,154.876
C08014=1061.535,-83.522,-62.649,171.449,26.075,154.876
C08015=1061.529,-83.772,-62.638,171.447,26.074,154.876
C08016=1061.523,-84.021,-62.627,171.445,26.072,154.876
C08017=1061.517,-84.271,-62.616,171.444,26.071,154.876
C08018=1061.510,-84.521,-62.606,171.442,26.070,154.876
C08019=1061.504,-84.770,-62.595,171.440,26.068,154.876
C08020=1061.498,-85.020,-62.583,171.439,26.067,154.876
C08021=1061.492,-85.270,-62.573,171.437,26.066,154.876
C08022=1061.486,-85.519,-62.562,171.435,26.064,154.876
C08023=1061.479,-85.769,-62.551,171.433,26.063,154.876
C08024=1061.473,-86.018,-62.541,171.432,26.062,154.876
C08025=1061.467,-86.268,-62.530,171.430,26.060,154.876
C08026=1061.461,-86.518,-62.519,171.428,26.059,154.876
C08027=1061.454,-86.767,-62.508,171.427,26.058,154.876
C08028=1061.449,-87.017,-62.498,171.425,26.056,154.875
C08029=1061.442,-87.267,-62.486,171.423,26.055,154.875
C08030=1061.436,-87.517,-62.477,171.421,26.053,154.875
C08031=1061.430,-87.766,-62.466,171.419,26.052,154.875
C08032=1061.424,-88.016,-62.455,171.417,26.050,154.875
C08033=1061.418,-88.266,-62.444,171.415,26.049,154.875
C08034=1061.412,-88.515,-62.433,171.414,26.048,154.875
C08035=1061.406,-88.765,-62.422,171.412,26.046,154.875
C08036=1061.399,-89.015,-62.412,171.410,26.045,154.875
C08037=1061.394,-89.265,-62.402,171.409,26.044,154.875
C08038=1061.387,-89.515,-62.391,171.407,26.043,154.875
C08039=1061.381,-89.764,-62.380,171.405,26.041,154.875
C08040=1061.375,-90.013,-62.369,171.403,26.040,154.875
C08041=1061.369,-90.263,-62.358,171.402,26.039,154.875
C08042=1061.363,-90.513,-62.349,171.400,26.037,154.875
C08043=1061.357,-90.763,-62.338,171.398,26.036,154.875
C08044=1061.350,-91.012,-62.327,171.397,26.034,154.875
C08045=1061.345,-91.262,-62.317,171.395,26.033,154.875
C08046=1061.338,-91.512,-62.305,171.392,26.032,154.875
C08047=1061.332,-91.762,-62.296,171.390,26.031,154.875
C08048=1061.326,-92.011,-62.285,171.389,26.029,154.875
C08049=1061.320,-92.260,-62.275,171.387,26.028,154.875
C08050=1061.314,-92.511,-62.264,171.385,26.026,154.874
C08051=1061.308,-92.761,-62.253,171.384,26.025,154.874
C08052=1061.302,-93.010,-62.243,171.382,26.024,154.874
C08053=1061.296,-93.259,-62.232,171.380,26.023,154.874
C08054=1061.290,-93.510,-62.221,171.379,26.021,154.874
C08055=1061.283,-93.759,-62.211,171.377,26.020,154.874
C08056=1061.278,-94.009,-62.200,171.375,26.019,154.874
C08057=1061.271,-94.259,-62.191,171.373,26.018,154.874
C08058=1061.266,-94.508,-62.180,171.372,26.017,154.874
C08059=1061.259,-94.757,-62.170,171.370,26.015,154.874
C08060=1061.253,-95.008,-62.159,171.368,26.014,154.874
C08061=1061.247,-95.258,-62.148,171.366,26.012,154.874
C08062=1061.241,-95.507,-62.138,171.365,26.011,154.874
C08063=1061.236,-95.757,-62.128,171.362,26.010,154.874
C08064=1061.229,-96.006,-62.117,171.360,26.009,154.874
C08065=1061.223,-96.256,-62.106,171.359,26.007,154.874
C08066=1061.217,-96.506,-62.096,171.357,26.006,154.874
C08067=1061.211,-96.755,-62.086,171.355,26.005,154.874
C08068=1061.205,-97.006,-62.076,171.353,26.004,154.874
C08069=1061.199,-97.255,-62.065,171.352,26.003,154.874
C08070=1061.193,-97.505,-62.055,171.350,26.002,154.874
C08071=1061.186,-97.755,-62.044,171.348,26.000,154.874
C08072=1061.180,-98.004,-62.034,171.346,25.999,154.874
C08073=1061.173,-98.289,-62.022,171.345,25.998,154.874
C08074=1061.166,-98.573,-62.010,171.342,25.997,154.874
C08075=1061.159,-98.858,-61.999,171.340,25.995,154.874
C08076=1061.152,-99.142,-61.987,171.339,25.994,154.874
C08077=1061.146,-99.392,-61.977,171.336,25.993,154.874
C08078=1061.140,-99.641,-61.967,171.334,25.992,154.874
C08079=1061.134,-99.891,-61.957,171.332,25.990,154.874
C08080=1061.128,-100.140,-61.947,171.331,25.989,154.874
C08081=1061.122,-100.390,-61.937,171.329,25.988,154.874
C08082=1061.116,-100.640,-61.926,171.327,25.987,154.874
C08083=1061.109,-100.890,-61.916,171.325,25.986,154.874
C08084=1061.103,-101.139,-61.906,171.324,25.984,154.874
C08085=1061.097,-101.389,-61.896,171.322,25.984,154.874
C08086=1061.091,-101.639,-61.886,171.320,25.983,154.874
C08087=1061.084,-101.888,-61.876,171.318,25.981,154.874
C08088=1061.079,-102.139,-61.866,171.317,25.980,154.874
C08089=1061.073,-102.388,-61.856,171.315,25.979,154.874
C08090=1061.066,-102.638,-61.846,171.313,25.978,154.874
C08091=1061.060,-102.888,-61.835,171.311,25.977,154.874
C08092=1061.054,-103.138,-61.825,171.309,25.976,154.874
C08093=1061.048,-103.387,-61.816,171.308,25.975,154.874
C08094=1061.042,-103.637,-61.805,171.305,25.974,154.874
C08095=1061.036,-103.887,-61.795,171.303,25.972,154.874
C08096=1061.029,-104.136,-61.785,171.302,25.971,154.874
C08097=1061.023,-104.386,-61.775,171.300,25.971,154.874
C08098=1061.018,-104.636,-61.765,171.298,25.969,154.874
C08099=1061.011,-104.885,-61.755,171.296,25.968,154.874
C08100=1061.005,-105.135,-61.745,171.294,25.967,154.874
C08101=1061.000,-105.385,-61.735,171.293,25.966,154.874
C08102=1060.993,-105.634,-61.725,171.291,25.965,154.874
C08103=1060.986,-105.884,-61.715,171.289,25.964,154.874
C08104=1060.980,-106.134,-61.705,171.287,25.963,154.874
C08105=1060.974,-106.384,-61.695,171.285,25.962,154.874
C08106=1060.968,-106.634,-61.685,171.284,25.961,154.874
C08107=1060.962,-106.883,-61.675,171.282,25.960,154.874
C08108=1060.956,-107.133,-61.666,171.280,25.959,154.874
C08109=1060.950,-107.383,-61.655,171.278,25.958,154.874
C08110=1060.944,-107.632,-61.645,171.277,25.957,154.874
C08111=1060.938,-107.882,-61.636,171.274,25.956,154.874
C08112=1060.932,-108.132,-61.626,171.272,25.955,154.874
C08113=1060.925,-108.381,-61.616,171.270,25.954,154.874
C08114=1060.919,-108.631,-61.606,171.269,25.953,154.874
C08115=1060.913,-108.881,-61.597,171.267,25.952,154.874
C08116=1060.907,-109.131,-61.587,171.265,25.951,154.874
C08117=1060.901,-109.380,-61.576,171.263,25.950,154.874
C08118=1060.895,-109.630,-61.567,171.261,25.949,154.874
C08119=1060.889,-109.880,-61.557,171.260,25.949,154.874
C08120=1060.882,-110.129,-61.548,171.258,25.947,154.874
C08121=1060.876,-110.379,-61.538,171.256,25.947,154.874
C08122=1060.870,-110.628,-61.528,171.254,25.946,154.874
C08123=1060.864,-110.878,-61.518,171.252,25.944,154.874
C08124=1060.857,-111.128,-61.509,171.251,25.944,154.875
C08125=1060.851,-111.378,-61.499,171.249,25.943,154.875
C08126=1060.846,-111.628,-61.489,171.247,25.942,154.875
C08127=1060.840,-111.878,-61.479,171.245,25.941,154.875
C08128=1060.834,-112.128,-61.470,171.242,25.940,154.875
C08129=1060.827,-112.377,-61.460,171.241,25.939,154.875
C08130=1060.821,-112.627,-61.450,171.239,25.938,154.875
C08131=1060.815,-112.876,-61.440,171.237,25.937,154.875
C08132=1060.809,-113.126,-61.431,171.235,25.936,154.875
C08133=1060.802,-113.376,-61.421,171.234,25.935,154.875
C08134=1060.796,-113.626,-61.412,171.232,25.935,154.875
C08135=1060.790,-113.876,-61.402,171.230,25.933,154.875
C08136=1060.784,-114.125,-61.393,171.228,25.933,154.875
C08137=1060.777,-114.408,-61.381,171.226,25.932,154.875
C08138=1060.770,-114.691,-61.370,171.224,25.931,154.875
C08139=1060.763,-114.973,-61.360,171.222,25.930,154.875
C08140=1060.756,-115.257,-61.349,171.220,25.929,154.875
C08141=1060.750,-115.507,-61.339,171.218,25.928,154.875
C08142=1060.744,-115.756,-61.330,171.216,25.927,154.875
C08143=1060.738,-116.006,-61.320,171.214,25.927,154.876
C08144=1060.732,-116.255,-61.311,171.213,25.925,154.875
C08145=1060.726,-116.505,-61.301,171.210,25.925,154.876
C08146=1060.720,-116.755,-61.292,171.208,25.923,154.876
C08147=1060.714,-117.005,-61.282,171.206,25.923,154.876
C08148=1060.707,-117.254,-61.272,171.204,25.922,154.876
C08149=1060.701,-117.504,-61.263,171.203,25.921,154.876
C08150=1060.694,-117.754,-61.254,171.201,25.920,154.876
C08151=1060.688,-118.004,-61.244,171.199,25.920,154.876
C08152=1060.682,-118.253,-61.235,171.197,25.919,154.876
C08153=1060.676,-118.503,-61.225,171.195,25.918,154.876
C08154=1060.670,-118.753,-61.216,171.194,25.918,154.876
C08155=1060.664,-119.002,-61.206,171.192,25.917,154.876
C08156=1060.658,-119.252,-61.197,171.190,25.916,154.876
C08157=1060.652,-119.502,-61.188,171.188,25.915,154.876
C08158=1060.646,-119.752,-61.178,171.186,25.915,154.876
C08159=1060.640,-120.002,-61.169,171.184,25.913,154.876
C08160=1060.634,-120.252,-61.159,171.183,25.913,154.877
C08161=1060.627,-120.501,-61.150,171.181,25.912,154.877
C08162=1060.620,-120.751,-61.141,171.179,25.912,154.877
C08163=1060.615,-121.000,-61.132,171.177,25.910,154.877
C08164=1060.609,-121.250,-61.122,171.174,25.910,154.877
C08165=1060.603,-121.500,-61.113,171.172,25.909,154.877
C08166=1060.597,-121.750,-61.104,171.171,25.908,154.877
C08167=1060.591,-122.000,-61.094,171.169,25.908,154.877
C08168=1060.584,-122.249,-61.085,171.167,25.907,154.877
C08169=1060.577,-122.499,-61.076,171.165,25.906,154.877
C08170=1060.572,-122.748,-61.066,171.163,25.905,154.877
C08171=1060.566,-122.999,-61.057,171.161,25.905,154.878
C08172=1060.560,-123.248,-61.048,171.160,25.904,154.878
C08173=1060.554,-123.498,-61.038,171.158,25.904,154.878
C08174=1060.547,-123.748,-61.029,171.156,25.902,154.878
C08175=1060.541,-123.998,-61.020,171.154,25.902,154.878
C08176=1060.535,-124.247,-61.011,171.152,25.901,154.878
C08177=1060.529,-124.497,-61.002,171.150,25.901,154.878
C08178=1060.523,-124.747,-60.992,171.148,25.900,154.878
C08179=1060.516,-124.996,-60.983,171.147,25.900,154.878
C08180=1060.510,-125.247,-60.974,171.145,25.899,154.878
C08181=1060.505,-125.496,-60.965,171.143,25.898,154.878
C08182=1060.498,-125.746,-60.956,171.141,25.898,154.879
C08183=1060.492,-125.996,-60.947,171.139,25.897,154.879
C08184=1060.486,-126.246,-60.938,171.137,25.897,154.879
C08185=1060.480,-126.495,-60.928,171.134,25.896,154.879
C08186=1060.474,-126.744,-60.919,171.133,25.895,154.879
C08187=1060.467,-126.995,-60.911,171.131,25.895,154.879
C08188=1060.461,-127.244,-60.901,171.129,25.894,154.879
C08189=1060.455,-127.494,-60.892,171.127,25.893,154.879
C08190=1060.448,-127.744,-60.883,171.125,25.893,154.879
C08191=1060.444,-127.994,-60.874,171.123,25.892,154.879
C08192=1060.439,-128.243,-60.863,171.122,25.890,154.879
C08193=1060.436,-128.494,-60.853,171.120,25.888,154.879
C08194=1060.435,-128.745,-60.841,171.119,25.886,154.879
C08195=1060.435,-128.996,-60.828,171.118,25.882,154.878
C08196=1060.436,-129.245,-60.816,171.117,25.879,154.878
C08197=1060.439,-129.498,-60.803,171.116,25.874,154.877
C08198=1060.443,-129.749,-60.788,171.115,25.869,154.876
C08199=1060.450,-130.000,-60.773,171.115,25.864,154.875
C08200=1060.456,-130.250,-60.757,171.115,25.858,154.874
C08201=1060.078,-130.273,-60.951,171.067,26.016,154.908
C08202=1060.071,-130.023,-60.966,171.067,26.022,154.909
C08203=1060.065,-129.772,-60.982,171.068,26.028,154.909
C08204=1060.061,-129.520,-60.996,171.069,26.032,154.910
C08205=1060.057,-129.269,-61.010,171.069,26.037,154.911
C08206=1060.056,-129.019,-61.023,171.070,26.040,154.911
C08207=1060.056,-128.768,-61.035,171.071,26.044,154.912
C08208=1060.057,-128.518,-61.047,171.073,26.046,154.912
C08209=1060.060,-128.267,-61.058,171.074,26.049,154.912
C08210=1060.064,-128.017,-61.068,171.076,26.050,154.912
C08211=1060.069,-127.766,-61.077,171.078,26.051,154.913
C08212=1060.076,-127.517,-61.086,171.080,26.052,154.912
C08213=1060.082,-127.267,-61.096,171.082,26.052,154.912
C08214=1060.087,-127.017,-61.104,171.084,26.053,154.912
C08215=1060.094,-126.768,-61.113,171.085,26.053,154.912
C08216=1060.100,-126.518,-61.123,171.087,26.054,154.912
C08217=1060.106,-126.268,-61.132,171.089,26.054,154.912
C08218=1060.112,-126.018,-61.141,171.091,26.055,154.912
C08219=1060.119,-125.769,-61.150,171.093,26.056,154.912
C08220=1060.125,-125.519,-61.160,171.095,26.056,154.912
C08221=1060.131,-125.269,-61.168,171.097,26.057,154.911
C08222=1060.137,-125.019,-61.178,171.098,26.057,154.911
C08223=1060.144,-124.770,-61.187,171.100,26.058,154.911
C08224=1060.149,-124.520,-61.195,171.102,26.058,154.911
C08225=1060.155,-124.270,-61.205,171.104,26.059,154.911
C08226=1060.161,-124.020,-61.215,171.107,26.060,154.911
C08227=1060.168,-123.771,-61.224,171.109,26.061,154.911
C08228=1060.174,-123.521,-61.233,171.110,26.062,154.911
C08229=1060.180,-123.271,-61.242,171.112,26.062,154.911
C08230=1060.186,-123.022,-61.251,171.114,26.063,154.911
C08231=1060.192,-122.772,-61.261,171.116,26.063,154.911
C08232=1060.198,-122.522,-61.270,171.118,26.064,154.910
C08233=1060.205,-122.272,-61.279,171.120,26.065,154.910
C08234=1060.211,-122.022,-61.288,171.122,26.066,154.910
C08235=1060.217,-121.772,-61.298,171.123,26.066,154.910
C08236=1060.223,-121.523,-61.307,171.125,26.067,154.910
C08237=1060.229,-121.273,-61.316,171.127,26.068,154.910
C08238=1060.235,-121.024,-61.326,171.129,26.069,154.910
C08239=1060.241,-120.774,-61.336,171.131,26.069,154.910
C08240=1060.247,-120.523,-61.344,171.133,26.070,154.910
C08241=1060.254,-120.274,-61.353,171.135,26.070,154.910
C08242=1060.260,-120.024,-61.363,171.136,26.071,154.910
C08243=1060.266,-119.775,-61.372,171.138,26.072,154.910
C08244=1060.272,-119.525,-61.382,171.141,26.073,154.910
C08245=1060.278,-119.275,-61.391,171.143,26.074,154.909
C08246=1060.284,-119.026,-61.401,171.145,26.075,154.909
C08247=1060.290,-118.776,-61.410,171.146,26.075,154.909
C08248=1060.297,-118.526,-61.420,171.148,26.076,154.909
C08249=1060.303,-118.276,-61.430,171.150,26.077,154.909
C08250=1060.309,-118.026,-61.439,171.152,26.078,154.909
C08251=1060.316,-117.777,-61.448,171.154,26.078,154.909
C08252=1060.322,-117.527,-61.458,171.156,26.079,154.909
C08253=1060.327,-117.277,-61.466,171.157,26.080,154.909
C08254=1060.333,-117.028,-61.476,171.159,26.081,154.909
C08255=1060.340,-116.778,-61.485,171.161,26.081,154.909
C08256=1060.346,-116.528,-61.495,171.163,26.082,154.909
C08257=1060.352,-116.278,-61.504,171.165,26.083,154.909
C08258=1060.358,-116.028,-61.514,171.167,26.084,154.909
C08259=1060.364,-115.779,-61.524,171.168,26.085,154.909
C08260=1060.371,-115.529,-61.533,171.170,26.085,154.909
C08261=1060.377,-115.279,-61.543,171.173,26.087,154.908
C08262=1060.383,-114.997,-61.554,171.175,26.087,154.908
C08263=1060.391,-114.713,-61.564,171.177,26.088,154.908
C08264=1060.397,-114.431,-61.576,171.179,26.089,154.908
C08265=1060.404,-114.148,-61.587,171.181,26.090,154.908
C08266=1060.410,-113.898,-61.596,171.183,26.091,154.908
C08267=1060.417,-113.648,-61.606,171.185,26.092,154.908
C08268=1060.423,-113.398,-61.615,171.187,26.093,154.908
C08269=1060.429,-113.148,-61.625,171.188,26.093,154.908
C08270=1060.435,-112.899,-61.635,171.190,26.095,154.908
C08271=1060.442,-112.649,-61.645,171.192,26.095,154.908
C08272=1060.448,-112.400,-61.654,171.194,26.096,154.908
C08273=1060.454,-112.150,-61.664,171.196,26.097,154.908
C08274=1060.460,-111.900,-61.674,171.197,26.098,154.908
C08275=1060.466,-111.650,-61.683,171.199,26.099,154.908
C08276=1060.472,-111.400,-61.693,171.202,26.100,154.908
C08277=1060.478,-111.150,-61.703,171.204,26.101,154.908
C08278=1060.484,-110.901,-61.713,171.206,26.102,154.908
C08279=1060.491,-110.651,-61.723,171.207,26.103,154.908
C08280=1060.497,-110.401,-61.732,171.209,26.104,154.908
C08281=1060.503,-110.152,-61.742,171.211,26.105,154.908
C08282=1060.509,-109.902,-61.751,171.213,26.105,154.907
C08283=1060.516,-109.653,-61.762,171.214,26.107,154.907
C08284=1060.522,-109.403,-61.771,171.216,26.107,154.907
C08285=1060.527,-109.153,-61.781,171.218,26.108,154.907
C08286=1060.533,-108.903,-61.791,171.220,26.110,154.907
C08287=1060.540,-108.653,-61.801,171.222,26.110,154.907
C08288=1060.546,-108.404,-61.811,171.223,26.111,154.907
C08289=1060.552,-108.154,-61.820,171.225,26.112,154.907
C08290=1060.558,-107.904,-61.830,171.227,26.113,154.907
C08291=1060.565,-107.655,-61.840,171.229,26.114,154.907
C08292=1060.571,-107.405,-61.850,171.232,26.115,154.907
C08293=1060.576,-107.155,-61.860,171.233,26.116,154.907
C08294=1060.583,-106.906,-61.870,171.235,26.117,154.907
C08295=1060.589,-106.656,-61.879,171.237,26.118,154.907
C08296=1060.595,-106.407,-61.889,171.239,26.119,154.907
C08297=1060.601,-106.156,-61.900,171.240,26.120,154.907
C08298=1060.607,-105.907,-61.909,171.242,26.122,154.907
C08299=1060.613,-105.657,-61.919,171.244,26.122,154.907
C08300=1060.620,-105.408,-61.929,171.246,26.123,154.907
C08301=1060.626,-105.157,-61.939,171.248,26.124,154.907
C08302=1060.632,-104.908,-61.950,171.249,26.126,154.907
C08303=1060.638,-104.658,-61.959,171.251,26.126,154.907
C08304=1060.644,-104.408,-61.969,171.253,26.127,154.907
C08305=1060.650,-104.159,-61.980,171.255,26.129,154.907
C08306=1060.656,-103.909,-61.989,171.256,26.130,154.907
C08307=1060.663,-103.660,-62.000,171.258,26.130,154.907
C08308=1060.668,-103.410,-62.010,171.261,26.132,154.907
C08309=1060.674,-103.160,-62.019,171.263,26.133,154.907
C08310=1060.681,-102.911,-62.030,171.264,26.134,154.907
C08311=1060.686,-102.660,-62.040,171.266,26.135,154.907
C08312=1060.693,-102.411,-62.050,171.268,26.136,154.907
C08313=1060.700,-102.161,-62.060,171.270,26.137,154.907
C08314=1060.705,-101.911,-62.070,171.272,26.138,154.907
C08315=1060.711,-101.661,-62.080,171.273,26.139,154.907
C08316=1060.718,-101.412,-62.090,171.275,26.141,154.907
C08317=1060.723,-101.162,-62.101,171.277,26.142,154.907
C08318=1060.730,-100.912,-62.110,171.279,26.143,154.907
C08319=1060.736,-100.663,-62.121,171.280,26.143,154.907
C08320=1060.742,-100.412,-62.131,171.282,26.145,154.907
C08321=1060.749,-100.163,-62.142,171.284,26.146,154.907
C08322=1060.755,-99.913,-62.151,171.286,26.147,154.907
C08323=1060.760,-99.664,-62.162,171.288,26.148,154.907
C08324=1060.767,-99.414,-62.172,171.290,26.150,154.907
C08325=1060.773,-99.165,-62.182,171.292,26.151,154.907
C08326=1060.780,-98.880,-62.194,171.294,26.152,154.907
C08327=1060.787,-98.596,-62.206,171.295,26.153,154.907
C08328=1060.794,-98.311,-62.217,171.298,26.155,154.907
C08329=1060.801,-98.027,-62.229,171.300,26.156,154.907
C08330=1060.807,-97.776,-62.239,171.302,26.157,154.907
C08331=1060.814,-97.527,-62.249,171.303,26.158,154.907
C08332=1060.819,-97.277,-62.259,171.305,26.159,154.907
C08333=1060.825,-97.027,-62.270,171.307,26.160,154.907
C08334=1060.831,-96.778,-62.280,171.309,26.162,154.907
C08335=1060.837,-96.528,-62.291,171.310,26.163,154.907
C08336=1060.844,-96.278,-62.301,171.312,26.164,154.907
C08337=1060.850,-96.028,-62.312,171.315,26.165,154.907
C08338=1060.856,-95.779,-62.322,171.316,26.167,154.907
C08339=1060.862,-95.529,-62.333,171.318,26.168,154.907
C08340=1060.867,-95.279,-62.343,171.320,26.169,154.907
C08341=1060.874,-95.030,-62.353,171.322,26.171,154.907
C08342=1060.880,-94.779,-62.364,171.323,26.172,154.907
C08343=1060.886,-94.530,-62.374,171.325,26.173,154.907
C08344=1060.892,-94.281,-62.385,171.327,26.174,154.907
C08345=1060.898,-94.031,-62.394,171.329,26.175,154.907
C08346=1060.904,-93.781,-62.405,171.330,26.176,154.907
C08347=1060.910,-93.531,-62.416,171.332,26.178,154.907
C08348=1060.917,-93.282,-62.427,171.334,26.179,154.908
C08349=1060.922,-93.032,-62.437,171.335,26.181,154.908
C08350=1060.929,-92.783,-62.447,171.337,26.182,154.908
C08351=1060.935,-92.533,-62.458,171.339,26.183,154.908
C08352=1060.940,-92.282,-62.469,171.341,26.184,154.908
C08353=1060.947,-92.033,-62.479,171.343,26.186,154.908
C08354=1060.953,-91.784,-62.490,171.345,26.187,154.908
C08355=1060.959,-91.534,-62.501,171.347,26.188,154.908
C08356=1060.965,-91.284,-62.511,171.348,26.190,154.908
C08357=1060.971,-91.034,-62.521,171.350,26.191,154.908
C08358=1060.977,-90.785,-62.532,171.352,26.192,154.908
C08359=1060.984,-90.535,-62.543,171.354,26.194,154.908
C08360=1060.989,-90.285,-62.554,171.355,26.195,154.908
C08361=1060.996,-90.036,-62.563,171.357,26.196,154.908
C08362=1061.001,-89.786,-62.574,171.359,26.197,154.908
C08363=1061.008,-89.536,-62.586,171.360,26.199,154.908
C08364=1061.014,-89.287,-62.596,171.362,26.200,154.908
C08365=1061.020,-89.037,-62.607,171.364,26.201,154.908
C08366=1061.027,-88.787,-62.617,171.366,26.202,154.908
C08367=1061.032,-88.537,-62.628,171.367,26.204,154.908
C08368=1061.038,-88.288,-62.638,171.369,26.205,154.908
C08369=1061.045,-88.038,-62.649,171.372,26.207,154.908
C08370=1061.051,-87.788,-62.660,171.374,26.208,154.908
C08371=1061.057,-87.539,-62.671,171.375,26.210,154.909
C08372=1061.063,-87.290,-62.681,171.377,26.211,154.909
C08373=1061.069,-87.040,-62.692,171.379,26.212,154.909
C08374=1061.075,-86.790,-62.703,171.380,26.214,154.909
C08375=1061.082,-86.540,-62.713,171.382,26.215,154.909
C08376=1061.088,-86.290,-62.724,171.384,26.216,154.909
C08377=1061.093,-86.041,-62.735,171.386,26.217,154.909
C08378=1061.101,-85.791,-62.746,171.387,26.219,154.909
C08379=1061.106,-85.541,-62.756,171.389,26.220,154.909
C08380=1061.112,-85.292,-62.767,171.391,26.221,154.909
C08381=1061.118,-85.042,-62.779,171.392,26.223,154.909
C08382=1061.125,-84.792,-62.789,171.394,26.224,154.909
C08383=1061.131,-84.543,-62.800,171.396,26.225,154.909
C08384=1061.137,-84.293,-62.811,171.397,26.227,154.909
C08385=1061.143,-84.044,-62.821,171.400,26.229,154.909
C08386=1061.150,-83.793,-62.832,171.402,26.230,154.909
C08387=1061.155,-83.544,-62.843,171.403,26.232,154.909
C08388=1061.162,-83.295,-62.854,171.405,26.233,154.909
C08389=1061.168,-83.045,-62.865,171.407,26.235,154.910
C08390=1061.175,-82.763,-62.877,171.409,26.236,154.910
C08391=1061.182,-82.480,-62.890,171.410,26.237,154.910
C08392=1061.189,-82.197,-62.902,171.413,26.239,154.910
C08393=1061.196,-81.916,-62.914,171.415,26.241,154.910
C08394=1061.202,-81.665,-62.925,171.416,26.242,154.910
C08395=1061.208,-81.416,-62.936,171.418,26.244,154.910
C08396=1061.215,-81.166,-62.946,171.420,26.245,154.910
C08397=1061.221,-80.917,-62.958,171.421,26.246,154.910
C08398=1061.228,-80.667,-62.969,171.423,26.248,154.910
C08399=1061.234,-80.418,-62.980,171.426,26.249,154.910
C08400=1061.240,-80.168,-62.990,171.427,26.251,154.910
C08401=1061.246,-79.918,-63.002,171.429,26.252,154.910
C08402=1061.252,-79.669,-63.013,171.431,26.254,154.910
C08403=1061.258,-79.418,-63.024,171.433,26.255,154.910
C08404=1061.264,-79.169,-63.035,171.434,26.257,154.911
C08405=1061.270,-78.919,-63.046,171.436,26.258,154.911
C08406=1061.276,-78.670,-63.057,171.438,26.260,154.911
C08407=1061.283,-78.420,-63.068,171.439,26.261,154.911
C08408=1061.289,-78.170,-63.079,171.441,26.262,154.911
C08409=1061.295,-77.921,-63.090,171.443,26.264,154.911
C08410=1061.301,-77.671,-63.101,171.444,26.265,154.911
C08411=1061.307,-77.421,-63.112,171.446,26.267,154.911
C08412=1061.314,-77.172,-63.124,171.448,26.268,154.911
C08413=1061.319,-76.922,-63.135,171.449,26.270,154.911
C08414=1061.326,-76.672,-63.146,171.451,26.272,154.912
C08415=1061.331,-76.423,-63.157,171.453,26.273,154.912
C08416=1061.338,-76.173,-63.169,171.454,26.275,154.912
C08417=1061.344,-75.923,-63.180,171.457,26.276,154.912
C08418=1061.350,-75.673,-63.191,171.459,26.278,154.912
C08419=1061.356,-75.424,-63.202,171.460,26.280,154.912
C08420=1061.362,-75.174,-63.214,171.462,26.281,154.912
C08421=1061.368,-74.925,-63.225,171.464,26.283,154.912
C08422=1061.375,-74.675,-63.236,171.465,26.284,154.912
C08423=1061.380,-74.425,-63.247,171.467,26.286,154.912
C08424=1061.387,-74.175,-63.259,171.469,26.287,154.912
C08425=1061.393,-73.926,-63.270,171.470,26.289,154.913
C08426=1061.399,-73.676,-63.281,171.472,26.290,154.913
C08427=1061.405,-73.427,-63.293,171.474,26.292,154.913
C08428=1061.411,-73.177,-63.304,171.475,26.294,154.913
C08429=1061.417,-72.927,-63.315,171.477,26.295,154.913
C08430=1061.423,-72.677,-63.327,171.479,26.297,154.913
C08431=1061.429,-72.428,-63.338,171.480,26.299,154.913
C08432=1061.435,-72.178,-63.349,171.482,26.300,154.913
C08433=1061.441,-71.929,-63.361,171.484,26.302,154.913
C08434=1061.447,-71.679,-63.372,171.485,26.304,154.914
C08435=1061.453,-71.429,-63.384,171.487,26.305,154.914
C08436=1061.459,-71.180,-63.395,171.489,26.307,154.914
C08437=1061.465,-70.930,-63.406,171.491,26.309,154.914
C08438=1061.471,-70.681,-63.418,171.493,26.311,154.914
C08439=1061.477,-70.430,-63.430,171.494,26.312,154.914
C08440=1061.483,-70.182,-63.442,171.496,26.314,154.914
C08441=1061.489,-69.931,-63.453,171.498,26.315,154.914
C08442=1061.495,-69.681,-63.464,171.499,26.317,154.915
C08443=1061.501,-69.432,-63.476,171.501,26.319,154.915
C08444=1061.507,-69.182,-63.487,171.503,26.321,154.915
C08445=1061.513,-68.933,-63.499,171.504,26.322,154.915
C08446=1061.519,-68.683,-63.510,171.506,26.324,154.915
C08447=1061.525,-68.434,-63.522,171.508,26.325,154.915
C08448=1061.531,-68.183,-63.534,171.509,26.327,154.915
C08449=1061.537,-67.934,-63.545,171.511,26.329,154.915
C08450=1061.543,-67.684,-63.557,171.513,26.331,154.916
C08451=1061.550,-67.435,-63.569,171.514,26.332,154.916
C08452=1061.555,-67.185,-63.580,171.516,26.334,154.916
C08453=1061.562,-66.935,-63.592,171.517,26.336,154.916
C08454=1061.568,-66.655,-63.604,171.520,26.338,154.916
C08455=1061.575,-66.375,-63.617,171.522,26.340,154.916
C08456=1061.582,-66.096,-63.631,171.523,26.341,154.916
C08457=1061.589,-65.816,-63.644,171.526,26.344,154.917
C08458=1061.595,-65.565,-63.655,171.527,26.346,154.917
C08459=1061.601,-65.316,-63.667,171.529,26.347,154.917
C08460=1061.607,-65.066,-63.678,171.531,26.349,154.917
C08461=1061.613,-64.817,-63.691,171.532,26.350,154.917
C08462=1061.619,-64.566,-63.702,171.534,26.352,154.917
C08463=1061.625,-64.317,-63.714,171.536,26.354,154.917
C08464=1061.632,-64.068,-63.726,171.537,26.356,154.917
C08465=1061.637,-63.818,-63.737,171.539,26.357,154.918
C08466=1061.644,-63.569,-63.749,171.541,26.359,154.918
C08467=1061.650,-63.319,-63.761,171.542,26.361,154.918
C08468=1061.655,-63.069,-63.773,171.544,26.363,154.918
C08469=1061.662,-62.820,-63.784,171.546,26.364,154.918
C08470=1061.668,-62.570,-63.796,171.547,26.366,154.918
C08471=1061.674,-62.321,-63.807,171.549,26.368,154.918
C08472=1061.680,-62.071,-63.820,171.550,26.370,154.919
C08473=1061.687,-61.821,-63.832,171.552,26.371,154.919
C08474=1061.692,-61.572,-63.843,171.554,26.373,154.919
C08475=1061.698,-61.322,-63.855,171.555,26.375,154.919
C08476=1061.705,-61.072,-63.867,171.557,26.377,154.919
C08477=1061.711,-60.822,-63.878,171.559,26.378,154.919
C08478=1061.717,-60.573,-63.891,171.560,26.380,154.919
C08479=1061.723,-60.323,-63.903,171.562,26.382,154.920
C08480=1061.730,-60.073,-63.914,171.563,26.384,154.920
C08481=1061.735,-59.824,-63.926,171.566,26.386,154.920
C08482=1061.742,-59.574,-63.938,171.568,26.388,154.920
C08483=1061.748,-59.325,-63.950,171.569,26.390,154.920
C08484=1061.754,-59.074,-63.962,171.571,26.391,154.920
C08485=1061.760,-58.825,-63.973,171.573,26.393,154.921
C08486=1061.767,-58.576,-63.985,171.574,26.395,154.921
C08487=1061.772,-58.326,-63.998,171.576,26.397,154.921
C08488=1061.779,-58.076,-64.010,171.577,26.398,154.921
C08489=1061.785,-57.827,-64.021,171.579,26.400,154.921
C08490=1061.791,-57.577,-64.033,171.581,26.402,154.921
C08491=1061.797,-57.327,-64.045,171.582,26.403,154.921
C08492=1061.804,-57.078,-64.057,171.584,26.405,154.922
C08493=1061.809,-56.829,-64.069,171.586,26.407,154.922
C08494=1061.816,-56.579,-64.081,171.587,26.409,154.922
C08495=1061.822,-56.328,-64.093,171.589,26.411,154.922
C08496=1061.828,-56.079,-64.105,171.590,26.413,154.922
C08497=1061.835,-55.829,-64.117,171.592,26.415,154.922
C08498=1061.840,-55.580,-64.129,171.594,26.416,154.923
C08499=1061.847,-55.331,-64.141,171.595,26.418,154.923
C08500=1061.854,-55.081,-64.153,171.597,26.420,154.923
C08501=1061.859,-54.831,-64.166,171.599,26.421,154.923
C08502=1061.866,-54.582,-64.178,171.600,26.423,154.923
C08503=1061.872,-54.331,-64.190,171.602,26.426,154.923
C08504=1061.878,-54.082,-64.201,171.603,26.427,154.923
C08505=1061.884,-53.833,-64.213,171.605,26.429,154.924
C08506=1061.894,-53.450,-64.232,171.608,26.432,154.924
C08507=1061.903,-53.067,-64.250,171.611,26.435,154.924
C08508=1061.913,-52.684,-64.269,171.613,26.438,154.924
C08509=1061.922,-52.301,-64.288,171.616,26.440,154.925
C08510=1061.929,-52.052,-64.300,171.617,26.442,154.925
C08511=1061.935,-51.802,-64.312,171.619,26.444,154.925
C08512=1061.941,-51.552,-64.324,171.621,26.446,154.925
C08513=1061.948,-51.303,-64.336,171.622,26.448,154.925
C08514=1061.958,-50.908,-64.355,171.625,26.450,154.925
C08515=1061.967,-50.513,-64.375,171.628,26.454,154.926
C08516=1061.978,-50.117,-64.394,171.630,26.457,154.926
C08517=1061.987,-49.722,-64.414,171.633,26.460,154.926
C08518=1061.993,-49.472,-64.426,171.634,26.461,154.926
C08519=1061.999,-49.223,-64.439,171.636,26.464,154.927
C08520=1062.005,-48.973,-64.451,171.638,26.466,154.927
C08521=1062.010,-48.723,-64.464,171.639,26.468,154.927
C08522=1062.017,-48.474,-64.476,171.641,26.470,154.927
C08523=1062.023,-48.224,-64.489,171.642,26.471,154.927
C08524=1062.029,-47.975,-64.501,171.644,26.474,154.928
C08525=1062.035,-47.726,-64.513,171.646,26.475,154.928
C08526=1062.041,-47.476,-64.526,171.647,26.478,154.928
C08527=1062.047,-47.226,-64.538,171.649,26.479,154.928
C08528=1062.053,-46.976,-64.551,171.650,26.482,154.928
C08529=1062.060,-46.726,-64.563,171.652,26.483,154.929
C08530=1062.066,-46.477,-64.576,171.654,26.485,154.929
C08531=1062.072,-46.227,-64.588,171.655,26.488,154.929
C08532=1062.078,-45.977,-64.601,171.657,26.489,154.929
C08533=1062.084,-45.728,-64.613,171.658,26.492,154.929
C08534=1062.090,-45.479,-64.625,171.660,26.493,154.930
C08535=1062.096,-45.229,-64.638,171.661,26.496,154.930
C08536=1062.102,-44.980,-64.651,171.663,26.497,154.930
C08537=1062.108,-44.730,-64.663,171.665,26.499,154.930
C08538=1062.114,-44.480,-64.675,171.666,26.501,154.930
C08539=1062.120,-44.230,-64.688,171.668,26.503,154.931
C08540=1062.126,-43.981,-64.701,171.669,26.505,154.931
C08541=1062.133,-43.731,-64.713,171.671,26.507,154.931
C08542=1062.139,-43.481,-64.726,171.673,26.509,154.931
C08543=1062.145,-43.232,-64.738,171.674,26.511,154.931
C08544=1062.151,-42.982,-64.752,171.676,26.514,154.932
C08545=1062.158,-42.733,-64.764,171.677,26.515,154.932
C08546=1062.164,-42.483,-64.776,171.679,26.518,154.932
C08547=1062.170,-42.234,-64.789,171.681,26.519,154.932
C08548=1062.176,-41.984,-64.802,171.682,26.522,154.932
C08549=1062.182,-41.735,-64.814,171.685,26.524,154.933
C08550=1062.188,-41.485,-64.826,171.686,26.526,154.933
C08551=1062.194,-41.236,-64.839,171.688,26.528,154.933
C08552=1062.200,-40.986,-64.852,171.689,26.530,154.933
C08553=1062.206,-40.736,-64.864,171.691,26.532,154.933
C08554=1062.213,-40.487,-64.877,171.693,26.534,154.934
C08555=1062.219,-40.237,-64.890,171.694,26.536,154.934
C08556=1062.225,-39.988,-64.903,171.696,26.538,154.934
C08557=1062.231,-39.738,-64.916,171.697,26.540,154.934
C08558=1062.237,-39.488,-64.928,171.699,26.542,154.934
C08559=1062.244,-39.239,-64.941,171.701,26.544,154.935
C08560=1062.250,-38.989,-64.953,171.702,26.546,154.935
C08561=1062.256,-38.739,-64.966,171.704,26.548,154.935
C08562=1062.262,-38.489,-64.980,171.705,26.550,154.935
C08563=1062.268,-38.239,-64.992,171.707,26.552,154.935
C08564=1062.274,-37.990,-65.005,171.708,26.554,154.936
C08565=1062.280,-37.740,-65.018,171.710,26.557,154.936
C08566=1062.287,-37.491,-65.031,171.712,26.558,154.936
C08567=1062.292,-37.242,-65.043,171.713,26.561,154.936
C08568=1062.298,-36.993,-65.057,171.715,26.563,154.937
C08569=1062.304,-36.743,-65.069,171.716,26.565,154.937
C08570=1062.310,-36.493,-65.082,171.718,26.567,154.937
C08571=1062.317,-36.243,-65.095,171.719,26.569,154.937
C08572=1062.323,-35.993,-65.108,171.721,26.571,154.937
C08573=1062.329,-35.744,-65.121,171.723,26.573,154.938
C08574=1062.335,-35.494,-65.134,171.724,26.576,154.938
C08575=1062.341,-35.245,-65.147,171.726,26.577,154.938
C08576=1062.347,-34.995,-65.160,171.727,26.580,154.938
C08577=1062.353,-34.745,-65.173,171.729,26.582,154.939
C08578=1062.359,-34.467,-65.188,171.730,26.584,154.939
C08579=1062.367,-34.189,-65.202,171.732,26.587,154.939
C08580=1062.373,-33.910,-65.216,171.733,26.589,154.939
C08581=1062.380,-33.632,-65.231,171.736,26.592,154.940
C08582=1062.386,-33.383,-65.244,171.738,26.593,154.940
C08583=1062.392,-33.133,-65.257,171.739,26.596,154.940
C08584=1062.398,-32.883,-65.270,171.741,26.598,154.940
C08585=1062.405,-32.634,-65.283,171.742,26.600,154.941
C08586=1062.411,-32.384,-65.296,171.744,26.602,154.941
C08587=1062.417,-32.135,-65.309,171.745,26.604,154.941
C08588=1062.422,-31.885,-65.322,171.747,26.607,154.941
C08589=1062.428,-31.636,-65.335,171.749,26.608,154.941
C08590=1062.434,-31.386,-65.349,171.750,26.611,154.942
C08591=1062.441,-31.136,-65.361,171.752,26.613,154.942
C08592=1062.447,-30.887,-65.375,171.753,26.615,154.942
C08593=1062.453,-30.637,-65.388,171.755,26.617,154.942
C08594=1062.459,-30.387,-65.401,171.756,26.619,154.943
C08595=1062.465,-30.138,-65.414,171.758,26.622,154.943
C08596=1062.472,-29.889,-65.427,171.759,26.624,154.943
C08597=1062.478,-29.639,-65.440,171.761,26.626,154.943
C08598=1062.484,-29.390,-65.453,171.763,26.628,154.944
C08599=1062.491,-29.140,-65.467,171.764,26.630,154.944
C08600=1062.497,-28.890,-65.480,171.765,26.632,154.944
C08601=1062.502,-28.640,-65.493,171.766,26.634,154.944
C08602=1062.508,-28.391,-65.506,171.768,26.636,154.945
C08603=1062.514,-28.142,-65.520,171.769,26.639,154.945
C08604=1062.520,-27.892,-65.532,171.771,26.641,154.945
C08605=1062.527,-27.642,-65.546,171.773,26.643,154.945
C08606=1062.533,-27.393,-65.559,171.774,26.645,154.946
C08607=1062.540,-27.143,-65.572,171.776,26.647,154.946
C08608=1062.546,-26.894,-65.586,171.777,26.649,154.946
C08609=1062.551,-26.644,-65.599,171.779,26.651,154.946
C08610=1062.557,-26.395,-65.612,171.780,26.654,154.946
C08611=1062.564,-26.145,-65.626,171.782,26.656,154.947
C08612=1062.570,-25.895,-65.639,171.784,26.658,154.947
C08613=1062.576,-25.646,-65.653,171.785,26.660,154.947
C08614=1062.582,-25.396,-65.665,171.787,26.663,154.948
C08615=1062.588,-25.147,-65.679,171.788,26.665,154.948
C08616=1062.593,-24.897,-65.692,171.790,26.667,154.948
C08617=1062.600,-24.647,-65.706,171.791,26.670,154.948
C08618=1062.606,-24.398,-65.719,171.793,26.672,154.949
C08619=1062.612,-24.148,-65.733,171.794,26.674,154.949
C08620=1062.618,-23.899,-65.746,171.796,26.676,154.949
C08621=1062.624,-23.649,-65.759,171.798,26.678,154.949
C08622=1062.629,-23.400,-65.773,171.799,26.681,154.950
C08623=1062.636,-23.150,-65.787,171.801,26.683,154.950
C08624=1062.642,-22.900,-65.800,171.802,26.685,154.950
C08625=1062.648,-22.651,-65.814,171.804,26.687,154.950
C08626=1062.654,-22.402,-65.827,171.805,26.690,154.951
C08627=1062.660,-22.152,-65.840,171.807,26.692,154.951
C08628=1062.666,-21.902,-65.854,171.808,26.694,154.951
C08629=1062.673,-21.653,-65.868,171.810,26.697,154.951
C08630=1062.679,-21.403,-65.881,171.811,26.699,154.952
C08631=1062.684,-21.154,-65.895,171.813,26.701,154.952
C08632=1062.691,-20.904,-65.908,171.815,26.704,154.952
C08633=1062.697,-20.655,-65.922,171.816,26.706,154.952
C08634=1062.703,-20.405,-65.936,171.818,26.708,154.953
C08635=1062.709,-20.156,-65.949,171.819,26.710,154.953
C08636=1062.715,-19.906,-65.963,171.821,26.712,154.953
C08637=1062.721,-19.656,-65.976,171.822,26.715,154.953
C08638=1062.728,-19.407,-65.990,171.824,26.717,154.954
C08639=1062.733,-19.157,-66.003,171.825,26.719,154.954
C08640=1062.740,-18.907,-66.017,171.827,26.721,154.954
C08641=1062.746,-18.658,-66.030,171.829,26.724,154.954
C08642=1062.752,-18.379,-66.046,171.830,26.726,154.955
C08643=1062.759,-18.100,-66.062,171.832,26.729,154.955
C08644=1062.766,-17.820,-66.076,171.833,26.731,154.955
C08645=1062.773,-17.541,-66.092,171.835,26.733,154.956
C08646=1062.779,-17.292,-66.105,171.836,26.736,154.956
C08647=1062.785,-17.043,-66.119,171.838,26.738,154.956
C08648=1062.791,-16.793,-66.133,171.839,26.740,154.956
C08649=1062.798,-16.543,-66.147,171.841,26.743,154.957
C08650=1062.804,-16.294,-66.160,171.842,26.745,154.957
C08651=1062.810,-16.045,-66.173,171.844,26.747,154.957
C08652=1062.816,-15.794,-66.188,171.845,26.750,154.958
C08653=1062.822,-15.545,-66.201,171.847,26.752,154.958
C08654=1062.828,-15.295,-66.215,171.849,26.754,154.958
C08655=1062.835,-15.046,-66.229,171.850,26.756,154.958
C08656=1062.840,-14.797,-66.243,171.852,26.759,154.959
C08657=1062.847,-14.547,-66.256,171.853,26.761,154.959
C08658=1062.853,-14.297,-66.270,171.855,26.764,154.959
C08659=1062.859,-14.048,-66.284,171.856,26.766,154.960
C08660=1062.864,-13.798,-66.298,171.858,26.769,154.960
C08661=1062.871,-13.549,-66.313,171.859,26.771,154.960
C08662=1062.877,-13.299,-66.326,171.861,26.773,154.960
C08663=1062.882,-13.050,-66.340,171.862,26.775,154.961
C08664=1062.888,-12.799,-66.354,171.864,26.778,154.961
C08665=1062.895,-12.551,-66.368,171.865,26.780,154.961
C08666=1062.900,-12.301,-66.382,171.867,26.783,154.962
C08667=1062.907,-12.051,-66.395,171.868,26.785,154.962
C08668=1062.913,-11.802,-66.409,171.870,26.787,154.962
C08669=1062.919,-11.553,-66.424,171.872,26.790,154.962
C08670=1062.925,-11.303,-66.437,171.872,26.792,154.963
C08671=1062.931,-11.053,-66.451,171.874,26.794,154.963
C08672=1062.936,-10.804,-66.465,171.875,26.796,154.963
C08673=1062.943,-10.554,-66.480,171.877,26.799,154.963
C08674=1062.949,-10.305,-66.493,171.878,26.802,154.964
C08675=1062.956,-10.055,-66.507,171.880,26.804,154.964
C08676=1062.962,-9.806,-66.522,171.881,26.806,154.964
C08677=1062.967,-9.556,-66.536,171.883,26.808,154.965
C08678=1062.974,-9.306,-66.549,171.884,26.811,154.965
C08679=1062.980,-9.057,-66.564,171.886,26.813,154.965
C08680=1062.986,-8.807,-66.578,171.888,26.815,154.965
C08681=1062.992,-8.558,-66.591,171.889,26.818,154.966
C08682=1062.998,-8.309,-66.606,171.891,26.820,154.966
C08683=1063.004,-8.058,-66.620,171.892,26.823,154.966
C08684=1063.010,-7.810,-66.634,171.894,26.825,154.967
C08685=1063.016,-7.560,-66.648,171.895,26.827,154.967
C08686=1063.022,-7.310,-66.662,171.897,26.830,154.967
C08687=1063.029,-7.061,-66.676,171.898,26.832,154.967
C08688=1063.034,-6.811,-66.690,171.900,26.835,154.968
C08689=1063.040,-6.562,-66.705,171.901,26.837,154.968
C08690=1063.047,-6.312,-66.719,171.903,26.839,154.968
C08691=1063.052,-6.063,-66.732,171.903,26.841,154.969
C08692=1063.059,-5.813,-66.747,171.905,26.844,154.969
C08693=1063.065,-5.564,-66.761,171.907,26.846,154.969
C08694=1063.071,-5.314,-66.776,171.908,26.849,154.970
C08695=1063.077,-5.064,-66.789,171.910,26.851,154.970
C08696=1063.083,-4.815,-66.804,171.911,26.853,154.970
C08697=1063.090,-4.565,-66.818,171.913,26.856,154.970
C08698=1063.096,-4.316,-66.833,171.914,26.858,154.971
C08699=1063.101,-4.066,-66.846,171.916,26.860,154.971
C08700=1063.109,-3.817,-66.861,171.917,26.863,154.971
C08701=1063.114,-3.567,-66.875,171.919,26.865,154.972
C08702=1063.120,-3.318,-66.890,171.920,26.868,154.972
C08703=1063.126,-3.068,-66.903,171.922,26.870,154.972
C08704=1063.132,-2.818,-66.918,171.923,26.873,154.973
C08705=1063.138,-2.569,-66.932,171.925,26.875,154.973
C08706=1063.145,-2.288,-66.949,171.926,26.878,154.973
C08707=1063.152,-2.007,-66.964,171.928,26.880,154.973
C08708=1063.158,-1.727,-66.981,171.929,26.883,154.974
C08709=1063.165,-1.447,-66.998,171.931,26.886,154.974
C08710=1063.171,-1.196,-67.012,171.932,26.888,154.974
C08711=1063.177,-0.947,-67.026,171.934,26.891,154.975
C08712=1063.183,-0.697,-67.041,171.935,26.894,154.975
C08713=1063.189,-0.448,-67.055,171.937,26.896,154.975
C08714=1063.194,-0.199,-67.070,171.938,26.899,154.976
C08715=1063.201,0.051,-67.084,171.940,26.901,154.976
C08716=1063.206,0.300,-67.099,171.941,26.903,154.976
C08717=1063.213,0.550,-67.114,171.943,26.906,154.977
C08718=1063.218,0.799,-67.127,171.944,26.908,154.977
C08719=1063.225,1.049,-67.142,171.946,26.911,154.977
C08720=1063.230,1.298,-67.157,171.947,26.914,154.978
C08721=1063.236,1.548,-67.171,171.949,26.916,154.978
C08722=1063.242,1.797,-67.186,171.950,26.918,154.978
C08723=1063.249,2.047,-67.201,171.951,26.921,154.979
C08724=1063.255,2.297,-67.215,171.953,26.923,154.979
C08725=1063.260,2.546,-67.230,171.954,26.926,154.979
C08726=1063.267,2.796,-67.244,171.956,26.928,154.980
C08727=1063.273,3.045,-67.259,171.957,26.930,154.980
C08728=1063.279,3.295,-67.273,171.959,26.933,154.980
C08729=1063.285,3.544,-67.288,171.960,26.936,154.980
C08730=1063.291,3.793,-67.303,171.962,26.938,154.981
C08731=1063.297,4.042,-67.317,171.963,26.941,154.981
C08732=1063.303,4.293,-67.332,171.965,26.943,154.981
C08733=1063.309,4.542,-67.346,171.966,26.945,154.982
C08734=1063.315,4.791,-67.361,171.968,26.948,154.982
C08735=1063.321,5.041,-67.376,171.969,26.950,154.982
C08736=1063.327,5.290,-67.391,171.970,26.952,154.983
C08737=1063.333,5.540,-67.405,171.971,26.955,154.983
C08738=1063.339,5.789,-67.419,171.973,26.958,154.983
C08739=1063.345,6.039,-67.434,171.975,26.960,154.984
C08740=1063.352,6.288,-67.449,171.976,26.963,154.984
C08741=1063.357,6.537,-67.464,171.978,26.965,154.984
C08742=1063.364,6.787,-67.479,171.979,26.968,154.985
C08743=1063.369,7.037,-67.493,171.981,26.970,154.985
C08744=1063.376,7.286,-67.508,171.982,26.972,154.985
C08745=1063.381,7.536,-67.523,171.984,26.975,154.986
C08746=1063.387,7.785,-67.538,171.985,26.978,154.986
C08747=1063.394,8.035,-67.553,171.987,26.980,154.986
C08748=1063.400,8.285,-67.568,171.988,26.983,154.986
C08749=1063.406,8.533,-67.582,171.989,26.985,154.987
C08750=1063.412,8.783,-67.597,171.990,26.988,154.987
C08751=1063.418,9.033,-67.611,171.992,26.990,154.987
C08752=1063.424,9.282,-67.626,171.993,26.992,154.988
C08753=1063.430,9.532,-67.641,171.995,26.995,154.988
C08754=1063.437,9.782,-67.656,171.996,26.997,154.988
C08755=1063.442,10.031,-67.671,171.998,27.000,154.989
C08756=1063.449,10.280,-67.685,172.000,27.002,154.989
C08757=1063.455,10.530,-67.700,172.001,27.005,154.989
C08758=1063.460,10.779,-67.716,172.003,27.008,154.990
C08759=1063.467,11.029,-67.731,172.004,27.010,154.990
C08760=1063.473,11.279,-67.746,172.006,27.012,154.990
C08761=1063.479,11.527,-67.760,172.007,27.015,154.991
C08762=1063.485,11.777,-67.775,172.008,27.017,154.991
C08763=1063.492,12.027,-67.790,172.009,27.019,154.991
C08764=1063.498,12.276,-67.805,172.011,27.022,154.992
C08765=1063.504,12.525,-67.820,172.012,27.024,154.992
C08766=1063.510,12.775,-67.834,172.014,27.027,154.992
C08767=1063.517,13.025,-67.849,172.015,27.030,154.993
C08768=1063.522,13.274,-67.865,172.017,27.032,154.993
C08769=1063.528,13.524,-67.880,172.018,27.035,154.993
C08770=1063.535,13.806,-67.897,172.020,27.038,154.994
C08771=1063.542,14.089,-67.913,172.021,27.040,154.994
C08772=1063.550,14.371,-67.930,172.023,27.043,154.994
C08773=1063.556,14.655,-67.948,172.025,27.046,154.995
C08774=1063.562,14.904,-67.963,172.026,27.048,154.995
C08775=1063.568,15.153,-67.978,172.027,27.051,154.995
C08776=1063.574,15.403,-67.993,172.029,27.054,154.996
C08777=1063.580,15.652,-68.008,172.030,27.056,154.996
C08778=1063.586,15.901,-68.023,172.032,27.059,154.996
C08779=1063.592,16.151,-68.039,172.033,27.061,154.997
C08780=1063.598,16.401,-68.054,172.035,27.064,154.997
C08781=1063.604,16.650,-68.068,172.036,27.066,154.997
C08782=1063.610,16.900,-68.084,172.038,27.069,154.998
C08783=1063.616,17.149,-68.099,172.040,27.071,154.998
C08784=1063.622,17.398,-68.114,172.041,27.074,154.998
C08785=1063.628,17.648,-68.130,172.043,27.076,154.999
C08786=1063.634,17.897,-68.145,172.043,27.079,154.999
C08787=1063.641,18.147,-68.160,172.045,27.081,154.999
C08788=1063.647,18.396,-68.176,172.046,27.084,155.000
C08789=1063.653,18.645,-68.190,172.048,27.086,155.000
C08790=1063.659,18.895,-68.205,172.049,27.089,155.000
C08791=1063.665,19.145,-68.221,172.051,27.091,155.001
C08792=1063.671,19.395,-68.236,172.052,27.094,155.001
C08793=1063.677,19.643,-68.251,172.054,27.097,155.001
C08794=1063.683,19.893,-68.267,172.055,27.099,155.002
C08795=1063.689,20.143,-68.282,172.057,27.102,155.002
C08796=1063.695,20.392,-68.298,172.057,27.104,155.002
C08797=1063.701,20.642,-68.313,172.059,27.107,155.003
C08798=1063.706,20.891,-68.328,172.060,27.109,155.003
C08799=1063.713,21.141,-68.343,172.062,27.112,155.003
C08800=1063.719,21.390,-68.359,172.063,27.114,155.004
C08801=1063.725,21.640,-68.374,172.065,27.117,155.004
C08802=1063.730,21.889,-68.389,172.066,27.120,155.004
C08803=1063.737,22.138,-68.405,172.068,27.122,155.005
C08804=1063.743,22.387,-68.420,172.070,27.125,155.005
C08805=1063.749,22.637,-68.436,172.071,27.128,155.005
C08806=1063.756,22.886,-68.451,172.073,27.130,155.006
C08807=1063.761,23.136,-68.466,172.073,27.132,155.006
C08808=1063.767,23.385,-68.482,172.075,27.135,155.007
C08809=1063.773,23.635,-68.498,172.076,27.138,155.007
C08810=1063.779,23.884,-68.512,172.078,27.140,155.007
C08811=1063.785,24.134,-68.529,172.079,27.143,155.007
C08812=1063.792,24.383,-68.544,172.081,27.145,155.008
C08813=1063.797,24.632,-68.560,172.082,27.148,155.008
C08814=1063.803,24.882,-68.575,172.084,27.151,155.009
C08815=1063.809,25.132,-68.590,172.085,27.153,155.009
C08816=1063.815,25.381,-68.606,172.087,27.156,155.009
C08817=1063.821,25.631,-68.621,172.087,27.158,155.010
C08818=1063.827,25.880,-68.638,172.089,27.161,155.010
C08819=1063.834,26.130,-68.652,172.090,27.163,155.010
C08820=1063.840,26.379,-68.669,172.092,27.166,155.011
C08821=1063.845,26.628,-68.683,172.093,27.169,155.011
C08822=1063.851,26.877,-68.700,172.095,27.171,155.011
C08823=1063.858,27.127,-68.715,172.096,27.174,155.012
C08824=1063.864,27.376,-68.731,172.098,27.176,155.012
C08825=1063.870,27.626,-68.746,172.099,27.179,155.012
C08826=1063.876,27.875,-68.762,172.101,27.182,155.013
C08827=1063.882,28.125,-68.778,172.102,27.184,155.013
C08828=1063.888,28.374,-68.793,172.103,27.186,155.013
C08829=1063.894,28.624,-68.809,172.105,27.189,155.014
C08830=1063.900,28.873,-68.824,172.106,27.192,155.014
C08831=1063.906,29.123,-68.840,172.108,27.194,155.014
C08832=1063.912,29.372,-68.856,172.109,27.197,155.015
C08833=1063.918,29.621,-68.872,172.111,27.199,155.015
C08834=1063.925,29.906,-68.889,172.112,27.202,155.015
C08835=1063.932,30.190,-68.907,172.114,27.206,155.016
C08836=1063.938,30.473,-68.926,172.115,27.209,155.016
C08837=1063.945,30.758,-68.943,172.116,27.211,155.017
C08838=1063.951,31.007,-68.959,172.118,27.214,155.017
C08839=1063.957,31.256,-68.975,172.120,27.217,155.017
C08840=1063.963,31.506,-68.990,172.121,27.219,155.018
C08841=1063.969,31.755,-69.007,172.123,27.222,155.018
C08842=1063.975,32.005,-69.023,172.124,27.224,155.018
C08843=1063.981,32.254,-69.038,172.126,27.227,155.019
C08844=1063.987,32.504,-69.054,172.127,27.230,155.019
C08845=1063.993,32.753,-69.070,172.129,27.232,155.020
C08846=1063.999,33.003,-69.086,172.130,27.235,155.020
C08847=1064.006,33.252,-69.102,172.131,27.237,155.020
C08848=1064.011,33.501,-69.118,172.132,27.240,155.021
C08849=1064.017,33.751,-69.133,172.134,27.243,155.021
C08850=1064.022,34.000,-69.149,172.135,27.245,155.021
C08851=1064.029,34.249,-69.165,172.137,27.248,155.022
C08852=1064.035,34.498,-69.181,172.138,27.251,155.022
C08853=1064.041,34.748,-69.197,172.140,27.253,155.022
C08854=1064.047,34.998,-69.213,172.141,27.256,155.023
C08855=1064.053,35.247,-69.229,172.143,27.259,155.023
C08856=1064.059,35.496,-69.245,172.144,27.261,155.023
C08857=1064.065,35.746,-69.260,172.145,27.264,155.024
C08858=1064.071,35.995,-69.277,172.146,27.266,155.024
C08859=1064.077,36.245,-69.293,172.148,27.269,155.025
C08860=1064.084,36.494,-69.309,172.149,27.272,155.025
C08861=1064.090,36.743,-69.325,172.151,27.274,155.025
C08862=1064.095,36.993,-69.340,172.153,27.277,155.026
C08863=1064.101,37.243,-69.357,172.154,27.280,155.026
C08864=1064.108,37.492,-69.372,172.156,27.282,155.026
C08865=1064.114,37.741,-69.389,172.157,27.285,155.027
C08866=1064.120,37.990,-69.405,172.159,27.287,155.027
C08867=1064.126,38.240,-69.421,172.159,27.289,155.027
C08868=1064.131,38.490,-69.437,172.161,27.292,155.028
C08869=1064.137,38.739,-69.453,172.162,27.295,155.028
C08870=1064.143,38.988,-69.469,172.164,27.298,155.029
C08871=1064.149,39.238,-69.485,172.165,27.300,155.029
C08872=1064.155,39.487,-69.502,172.167,27.303,155.029
C08873=1064.161,39.736,-69.518,172.168,27.306,155.030
C08874=1064.167,39.986,-69.534,172.170,27.309,155.030
C08875=1064.173,40.235,-69.550,172.171,27.311,155.030
C08876=1064.179,40.484,-69.567,172.172,27.314,155.031
C08877=1064.185,40.734,-69.583,172.173,27.316,155.031
C08878=1064.191,40.984,-69.600,172.175,27.319,155.031
C08879=1064.197,41.233,-69.616,172.176,27.321,155.032
C08880=1064.203,41.482,-69.632,172.178,27.324,155.032
C08881=1064.209,41.732,-69.648,172.179,27.327,155.033
C08882=1064.215,41.982,-69.664,172.181,27.329,155.033
C08883=1064.221,42.231,-69.680,172.182,27.332,155.033
C08884=1064.227,42.480,-69.696,172.184,27.335,155.034
C08885=1064.233,42.730,-69.713,172.184,27.338,155.034
C08886=1064.239,42.979,-69.729,172.186,27.340,155.034
C08887=1064.245,43.229,-69.745,172.188,27.343,155.035
C08888=1064.251,43.478,-69.761,172.189,27.346,155.035
C08889=1064.257,43.727,-69.778,172.191,27.348,155.035
C08890=1064.263,43.976,-69.795,172.192,27.351,155.036
C08891=1064.269,44.225,-69.811,172.194,27.353,155.036
C08892=1064.275,44.475,-69.827,172.195,27.356,155.037
C08893=1064.280,44.724,-69.844,172.197,27.359,155.037
C08894=1064.286,44.974,-69.860,172.198,27.362,155.037
C08895=1064.292,45.223,-69.877,172.199,27.364,155.038
C08896=1064.298,45.473,-69.893,172.200,27.367,155.038
C08897=1064.304,45.723,-69.910,172.202,27.370,155.038
C08898=1064.311,46.007,-69.928,172.203,27.373,155.039
C08899=1064.318,46.290,-69.947,172.205,27.376,155.039
C08900=1064.324,46.574,-69.966,172.207,27.379,155.040
C08901=1064.331,46.859,-69.985,172.208,27.382,155.040
C08902=1064.337,47.108,-70.001,172.210,27.385,155.041
C08903=1064.342,47.357,-70.018,172.212,27.387,155.041
C08904=1064.348,47.606,-70.035,172.212,27.390,155.041
C08905=1064.354,47.856,-70.051,172.214,27.393,155.042
C08906=1064.360,48.105,-70.067,172.215,27.396,155.042
C08907=1064.365,48.355,-70.084,172.217,27.398,155.043
C08908=1064.372,48.603,-70.101,172.218,27.401,155.043
C08909=1064.377,48.853,-70.117,172.220,27.403,155.043
C08910=1064.384,49.103,-70.134,172.221,27.406,155.044
C08911=1064.389,49.352,-70.151,172.223,27.409,155.044
C08912=1064.395,49.602,-70.167,172.224,27.412,155.044
C08913=1064.401,49.850,-70.184,172.225,27.414,155.045
C08914=1064.407,50.100,-70.200,172.226,27.417,155.045
C08915=1064.413,50.349,-70.217,172.228,27.420,155.045
C08916=1064.419,50.599,-70.233,172.229,27.422,155.046
C08917=1064.425,50.848,-70.251,172.231,27.425,155.046
C08918=1064.431,51.098,-70.267,172.232,27.427,155.047
C08919=1064.437,51.347,-70.284,172.234,27.430,155.047
C08920=1064.443,51.596,-70.301,172.235,27.433,155.047
C08921=1064.449,51.845,-70.317,172.237,27.436,155.048
C08922=1064.454,52.095,-70.334,172.238,27.439,155.048
C08923=1064.461,52.345,-70.351,172.239,27.441,155.048
C08924=1064.467,52.594,-70.368,172.241,27.444,155.049
C08925=1064.473,52.843,-70.384,172.242,27.446,155.049
C08926=1064.478,53.093,-70.401,172.244,27.449,155.050
C08927=1064.484,53.342,-70.418,172.245,27.452,155.050
C08928=1064.491,53.592,-70.434,172.247,27.454,155.050
C08929=1064.496,53.841,-70.451,172.248,27.457,155.051
C08930=1064.502,54.090,-70.468,172.250,27.460,155.051
C08931=1064.508,54.339,-70.484,172.251,27.463,155.051
C08932=1064.514,54.588,-70.502,172.252,27.465,155.052
C08933=1064.520,54.838,-70.518,172.253,27.468,155.052
C08934=1064.526,55.088,-70.535,172.255,27.470,155.053
C08935=1064.532,55.336,-70.552,172.256,27.473,155.053
C08936=1064.538,55.586,-70.569,172.258,27.476,155.053
C08937=1064.545,55.836,-70.586,172.259,27.478,155.054
C08938=1064.550,56.085,-70.602,172.261,27.481,155.054
C08939=1064.556,56.335,-70.619,172.262,27.484,155.054
C08940=1064.562,56.583,-70.636,172.264,27.487,155.055
C08941=1064.569,56.833,-70.653,172.265,27.490,155.055
C08942=1064.574,57.082,-70.670,172.266,27.492,155.056
C08943=1064.580,57.332,-70.686,172.268,27.494,155.056
C08944=1064.586,57.580,-70.703,172.269,27.497,155.056
C08945=1064.592,57.831,-70.721,172.271,27.500,155.057
C08946=1064.598,58.080,-70.738,172.272,27.502,155.057
C08947=1064.604,58.329,-70.754,172.274,27.505,155.057
C08948=1064.610,58.579,-70.772,172.275,27.508,155.058
C08949=1064.616,58.828,-70.788,172.277,27.511,155.058
C08950=1064.623,59.077,-70.805,172.278,27.513,155.058
C08951=1064.628,59.327,-70.822,172.280,27.516,155.059
C08952=1064.635,59.576,-70.839,172.280,27.518,155.059
C08953=1064.640,59.825,-70.856,172.282,27.521,155.060
C08954=1064.646,60.074,-70.873,172.283,27.523,155.060
C08955=1064.653,60.324,-70.890,172.285,27.526,155.060
C08956=1064.658,60.573,-70.907,172.286,27.529,155.061
C08957=1064.665,60.823,-70.925,172.288,27.532,155.061
C08958=1064.671,61.072,-70.941,172.290,27.534,155.061
C08959=1064.677,61.321,-70.958,172.291,27.537,155.062
C08960=1064.683,61.571,-70.976,172.293,27.540,155.062
C08961=1064.689,61.820,-70.993,172.294,27.543,155.063
C08962=1064.695,62.104,-71.012,172.296,27.545,155.063
C08963=1064.702,62.387,-71.031,172.297,27.548,155.063
C08964=1064.710,62.672,-71.051,172.299,27.551,155.064
C08965=1064.716,62.955,-71.070,172.300,27.554,155.064
C08966=1064.723,63.204,-71.087,172.302,27.557,155.065
C08967=1064.729,63.454,-71.104,172.303,27.559,155.065
C08968=1064.735,63.703,-71.121,172.305,27.562,155.065
C08969=1064.741,63.952,-71.138,172.306,27.564,155.066
C08970=1064.747,64.202,-71.156,172.308,27.567,155.066
C08971=1064.753,64.451,-71.173,172.309,27.570,155.066
C08972=1064.759,64.701,-71.191,172.311,27.573,155.067
C08973=1064.765,64.949,-71.207,172.312,27.576,155.067
C08974=1064.771,65.199,-71.224,172.313,27.578,155.068
C08975=1064.777,65.449,-71.242,172.314,27.581,155.068
C08976=1064.783,65.697,-71.259,172.316,27.583,155.068
C08977=1064.788,65.947,-71.276,172.317,27.586,155.069
C08978=1064.795,66.197,-71.293,172.319,27.589,155.069
C08979=1064.801,66.446,-71.311,172.320,27.592,155.070
C08980=1064.806,66.695,-71.329,172.322,27.594,155.070
C08981=1064.813,66.944,-71.346,172.324,27.597,155.070
C08982=1064.818,67.194,-71.363,172.325,27.600,155.071
C08983=1064.824,67.443,-71.381,172.327,27.602,155.071
C08984=1064.831,67.692,-71.398,172.328,27.605,155.071
C08985=1064.836,67.941,-71.415,172.329,27.608,155.072
C08986=1064.842,68.191,-71.433,172.330,27.610,155.072
C08987=1064.848,68.440,-71.449,172.332,27.613,155.073
C08988=1064.854,68.690,-71.467,172.333,27.616,155.073
C08989=1064.860,68.939,-71.485,172.335,27.618,155.073
C08990=1064.866,69.188,-71.502,172.336,27.621,155.074
C08991=1064.872,69.438,-71.520,172.338,27.624,155.074
C08992=1064.878,69.687,-71.537,172.340,27.626,155.074
C08993=1064.885,69.936,-71.555,172.341,27.629,155.075
C08994=1064.890,70.185,-71.572,172.343,27.632,155.075
C08995=1064.896,70.435,-71.590,172.344,27.635,155.076
C08996=1064.901,70.684,-71.607,172.345,27.637,155.076
C08997=1064.907,70.933,-71.625,172.346,27.640,155.076
C08998=1064.914,71.183,-71.642,172.348,27.643,155.077
C08999=1064.919,71.432,-71.660,172.349,27.646,155.077
C09000=1064.925,71.682,-71.677,172.351,27.648,155.077
C09001=1064.931,71.931,-71.695,172.352,27.651,155.078
C09002=1064.937,72.180,-71.713,172.354,27.654,155.078
C09003=1064.943,72.429,-71.730,172.355,27.656,155.079
C09004=1064.949,72.678,-71.748,172.357,27.659,155.079
C09005=1064.955,72.928,-71.765,172.358,27.662,155.079
C09006=1064.961,73.177,-71.783,172.360,27.665,155.080
C09007=1064.967,73.427,-71.801,172.360,27.667,155.080
C09008=1064.972,73.676,-71.819,172.362,27.670,155.081
C09009=1064.979,73.925,-71.836,172.364,27.672,155.081
C09010=1064.985,74.174,-71.853,172.365,27.675,155.081
C09011=1064.991,74.424,-71.871,172.367,27.678,155.082
C09012=1064.996,74.673,-71.889,172.368,27.681,155.082
C09013=1065.002,74.923,-71.907,172.370,27.684,155.083
C09014=1065.008,75.172,-71.924,172.371,27.686,155.083
C09015=1065.014,75.422,-71.942,172.373,27.689,155.083
C09016=1065.020,75.670,-71.959,172.374,27.691,155.084
C09017=1065.026,75.920,-71.977,172.376,27.694,155.084
C09018=1065.032,76.168,-71.996,172.377,27.697,155.084
C09019=1065.038,76.418,-72.013,172.378,27.700,155.085
C09020=1065.044,76.667,-72.031,172.379,27.702,155.085
C09021=1065.050,76.917,-72.049,172.381,27.705,155.086
C09022=1065.055,77.166,-72.067,172.383,27.707,155.086
C09023=1065.062,77.416,-72.084,172.384,27.710,155.086
C09024=1065.067,77.665,-72.102,172.386,27.713,155.087
C09025=1065.074,77.914,-72.119,172.387,27.716,155.087
C09026=1065.080,78.198,-72.140,172.389,27.719,155.088
C09027=1065.087,78.481,-72.161,172.390,27.722,155.088
C09028=1065.094,78.765,-72.180,172.393,27.725,155.088
C09029=1065.100,79.048,-72.201,172.394,27.728,155.089
C09030=1065.107,79.298,-72.219,172.396,27.731,155.089
C09031=1065.112,79.547,-72.237,172.397,27.733,155.090
C09032=1065.119,79.796,-72.255,172.398,27.736,155.090
C09033=1065.123,80.046,-72.273,172.399,27.739,155.090
C09034=1065.129,80.295,-72.291,172.401,27.742,155.091
C09035=1065.135,80.544,-72.309,172.402,27.744,155.091
C09036=1065.141,80.793,-72.328,172.404,27.747,155.092
C09037=1065.147,81.042,-72.345,172.405,27.750,155.092
C09038=1065.153,81.292,-72.363,172.407,27.753,155.092
C09039=1065.159,81.541,-72.381,172.408,27.756,155.093
C09040=1065.165,81.790,-72.399,172.410,27.758,155.093
C09041=1065.170,82.039,-72.417,172.412,27.761,155.094
C09042=1065.177,82.289,-72.435,172.413,27.764,155.094
C09043=1065.182,82.538,-72.454,172.415,27.767,155.094
C09044=1065.188,82.788,-72.472,172.416,27.770,155.095
C09045=1065.194,83.037,-72.489,172.417,27.772,155.095
C09046=1065.200,83.286,-72.508,172.418,27.774,155.096
C09047=1065.206,83.536,-72.526,172.420,27.777,155.096
C09048=1065.211,83.785,-72.543,172.421,27.780,155.096
C09049=1065.218,84.034,-72.562,172.423,27.783,155.097
C09050=1065.224,84.283,-72.580,172.424,27.786,155.097
C09051=1065.229,84.533,-72.598,172.426,27.788,155.098
C09052=1065.235,84.782,-72.617,172.427,27.791,155.098
C09053=1065.241,85.031,-72.634,172.429,27.794,155.098
C09054=1065.247,85.280,-72.653,172.431,27.796,155.099
C09055=1065.253,85.530,-72.671,172.432,27.799,155.099
C09056=1065.259,85.779,-72.688,172.434,27.802,155.099
C09057=1065.265,86.028,-72.707,172.435,27.805,155.100
C09058=1065.270,86.277,-72.725,172.437,27.807,155.100
C09059=1065.276,86.526,-72.744,172.438,27.810,155.101
C09060=1065.282,86.776,-72.762,172.439,27.813,155.101
C09061=1065.288,87.025,-72.780,172.440,27.815,155.101
C09062=1065.294,87.274,-72.798,172.442,27.818,155.102
C09063=1065.301,87.524,-72.816,172.444,27.820,155.102
C09064=1065.306,87.773,-72.835,172.445,27.823,155.103
C09065=1065.312,88.023,-72.853,172.447,27.826,155.103
C09066=1065.318,88.272,-72.871,172.448,27.829,155.103
C09067=1065.324,88.521,-72.889,172.450,27.832,155.104
C09068=1065.330,88.770,-72.908,172.451,27.834,155.104
C09069=1065.336,89.020,-72.926,172.453,27.837,155.104
C09070=1065.341,89.268,-72.944,172.454,27.839,155.105
C09071=1065.348,89.517,-72.963,172.456,27.842,155.105
C09072=1065.354,89.767,-72.981,172.457,27.845,155.106
C09073=1065.360,90.016,-73.000,172.459,27.848,155.106
C09074=1065.366,90.265,-73.017,172.461,27.851,155.106
C09075=1065.372,90.515,-73.036,172.462,27.853,155.107
C09076=1065.378,90.765,-73.054,172.464,27.856,155.107
